LIN {X 0,Y 391.58,Z 838.555,A -85,B 0,C 180,E1 -11591.925,E2 -11591.925} C_VEL
LIN {X 0,Y 392.931,Z 851.436,A -85,B 0,C 180,E1 -11592.757,E2 -11592.757} C_VEL
LIN {X 0,Y 393.603,Z 859.87,A -85,B 0,C 180,E1 -11593.4,E2 -11593.4} C_VEL
LIN {X 0,Y 392.572,Z 872.076,A -85,B 0,C 180,E1 -11594.423,E2 -11594.423} C_VEL
LIN {X 0,Y 391.606,Z 884.787,A -85,B 0,C 180,E1 -11595.726,E2 -11595.726} C_VEL
LIN {X 0,Y 390.818,Z 894.925,A -85,B 0,C 180,E1 -11597.01,E2 -11597.01} C_VEL
LIN {X 0,Y 390.076,Z 904.821,A -85,B 0,C 180,E1 -11598.569,E2 -11598.569} C_VEL
LIN {X 0,Y 389.501,Z 912.81,A -85,B 0,C 180,E1 -11600.13,E2 -11600.13} C_VEL
LIN {X 0,Y 389.129,Z 919.186,A -85,B 0,C 180,E1 -11601.692,E2 -11601.692} C_VEL
LIN {X 0,Y 388.914,Z 924.388,A -85,B 0,C 180,E1 -11603.307,E2 -11603.307} C_VEL
LIN {X 0,Y 388.848,Z 928.132,A -85,B 0,C 180,E1 -11604.815,E2 -11604.815} C_VEL
LIN {X 0,Y 388.745,Z 930.111,A -85,B 0,C 180,E1 -11605.853,E2 -11605.853} C_VEL
LIN {X 0,Y 388.737,Z 931.665,A -85,B 0,C 180,E1 -11606.891,E2 -11606.891} C_VEL
LIN {X 0,Y 388.832,Z 932.76,A -85,B 0,C 180,E1 -11607.928,E2 -11607.928} C_VEL
LIN {X 0,Y 388.809,Z 933.409,A -85,B 0,C 180,E1 -11608.964,E2 -11608.964} C_VEL
LIN {X 0,Y 388.823,Z 933.651,A -85,B 0,C 180,E1 -11610,E2 -11610} C_VEL
LIN {X 0,Y 388.809,Z 933.483,A -85,B 0,C 180,E1 -11611.036,E2 -11611.036} C_VEL
LIN {X 0,Y 388.836,Z 932.855,A -85,B 0,C 180,E1 -11612.072,E2 -11612.072} C_VEL
LIN {X 0,Y 388.757,Z 930.333,A -85,B 0,C 180,E1 -11614.147,E2 -11614.147} C_VEL
LIN {X 0,Y 388.817,Z 926.891,A -85,B 0,C 180,E1 -11615.88,E2 -11615.88} C_VEL
LIN {X 0,Y 388.95,Z 923.164,A -85,B 0,C 180,E1 -11617.267,E2 -11617.267} C_VEL
LIN {X 0,Y 389.305,Z 916.887,A -85,B 0,C 180,E1 -11619.089,E2 -11619.089} C_VEL
LIN {X 0,Y 389.747,Z 910.033,A -85,B 0,C 180,E1 -11620.651,E2 -11620.651} C_VEL
LIN {X 0,Y 390.464,Z 901.593,A -85,B 0,C 180,E1 -11622.21,E2 -11622.21} C_VEL
LIN {X 0,Y 391.331,Z 891.841,A -85,B 0,C 180,E1 -11623.68,E2 -11623.68} C_VEL
LIN {X 0,Y 392.274,Z 880.534,A -85,B 0,C 180,E1 -11625.057,E2 -11625.057} C_VEL
LIN {X 0,Y 393.418,Z 868.68,A -85,B 0,C 180,E1 -11626.208,E2 -11626.208} C_VEL
LIN {X 0,Y 394.056,Z 859.025,A -85,B 0,C 180,E1 -11626.981,E2 -11626.981} C_VEL
LIN {X 0,Y 393.075,Z 845.103,A -85,B 0,C 180,E1 -11627.969,E2 -11627.969} C_VEL
LIN {X 0,Y 391.432,Z 832.806,A -85,B 0,C 180,E1 -11628.703,E2 -11628.703} C_VEL
LIN {X 0,Y 389.433,Z 823.338,A -85,B 0,C 180,E1 -11629.23,E2 -11629.23} C_VEL
LIN {X 0,Y 389.856,Z 815.289,A -85,B 0,C 180,E1 -11632.716,E2 -11632.716} C_VEL
LIN {X 0,Y 390.344,Z 808.49,A -85,B 0,C 180,E1 -11635.81,E2 -11635.81} C_VEL
LIN {X 0,Y 390.913,Z 801.858,A -85,B 0,C 180,E1 -11639.04,E2 -11639.04} C_VEL
LIN {X 0,Y 391.767,Z 795.266,A -85,B 0,C 180,E1 -11642.56,E2 -11642.56} C_VEL
LIN {X 0,Y 392.323,Z 791.243,A -85,B 0,C 180,E1 -11644.977,E2 -11644.977} C_VEL
LIN {X 0,Y 392.483,Z 787.628,A -85,B 0,C 180,E1 -11647.505,E2 -11647.505} C_VEL
LIN {X 0,Y 392.083,Z 784.529,A -85,B 0,C 180,E1 -11650.188,E2 -11650.188} C_VEL
LIN {X 0,Y 391.699,Z 782.043,A -85,B 0,C 180,E1 -11652.985,E2 -11652.985} C_VEL
LIN {X 0,Y 391.348,Z 780.234,A -85,B 0,C 180,E1 -11655.918,E2 -11655.918} C_VEL
LIN {X 0,Y 391.117,Z 779.149,A -85,B 0,C 180,E1 -11658.999,E2 -11658.999} C_VEL
LIN {X 0,Y 391.069,Z 778.836,A -85,B 0,C 180,E1 -11661.023,E2 -11661.023} C_VEL
LIN {X 0,Y 390.893,Z 778.937,A -85,B 0,C 180,E1 -11664.006,E2 -11664.006} C_VEL
LIN {X 0,Y 390.778,Z 779.326,A -85,B 0,C 180,E1 -11666.114,E2 -11666.114} C_VEL
LIN {X 0,Y 390.508,Z 780.09,A -85,B 0,C 180,E1 -11668.538,E2 -11668.538} C_VEL
LIN {X 0,Y 390.157,Z 781.62,A -85,B 0,C 180,E1 -11672.072,E2 -11672.072} C_VEL
LIN {X 0,Y 389.86,Z 783.496,A -85,B 0,C 180,E1 -11675.504,E2 -11675.504} C_VEL
LIN {X 0,Y 389.639,Z 785.619,A -85,B 0,C 180,E1 -11678.853,E2 -11678.853} C_VEL
LIN {X 0,Y 389.514,Z 787.117,A -85,B 0,C 180,E1 -11680.962,E2 -11680.962} C_VEL
LIN {X 0,Y 393.71,Z 799.562,A -85,B 0,C 180,E1 -11681.858,E2 -11681.858} C_VEL
LIN {X 0,Y 395.904,Z 808.974,A -85,B 0,C 180,E1 -11682.582,E2 -11682.582} C_VEL
LIN {X 0,Y 394.972,Z 821.103,A -85,B 0,C 180,E1 -11683.458,E2 -11683.458} C_VEL
LIN {X 0,Y 394.076,Z 832.258,A -85,B 0,C 180,E1 -11684.483,E2 -11684.483} C_VEL
LIN {X 0,Y 393.023,Z 843.465,A -85,B 0,C 180,E1 -11685.765,E2 -11685.765} C_VEL
LIN {X 0,Y 392.055,Z 852.61,A -85,B 0,C 180,E1 -11687.05,E2 -11687.05} C_VEL
LIN {X 0,Y 391.22,Z 861.469,A -85,B 0,C 180,E1 -11688.602,E2 -11688.602} C_VEL
LIN {X 0,Y 390.495,Z 868.618,A -85,B 0,C 180,E1 -11690.154,E2 -11690.154} C_VEL
LIN {X 0,Y 389.9,Z 874.374,A -85,B 0,C 180,E1 -11691.708,E2 -11691.708} C_VEL
LIN {X 0,Y 389.555,Z 878.773,A -85,B 0,C 180,E1 -11693.215,E2 -11693.215} C_VEL
LIN {X 0,Y 389.112,Z 882.348,A -85,B 0,C 180,E1 -11694.818,E2 -11694.818} C_VEL
LIN {X 0,Y 389.158,Z 884.056,A -85,B 0,C 180,E1 -11695.856,E2 -11695.856} C_VEL
LIN {X 0,Y 389.016,Z 885.331,A -85,B 0,C 180,E1 -11696.892,E2 -11696.892} C_VEL
LIN {X 0,Y 388.923,Z 886.208,A -85,B 0,C 180,E1 -11697.928,E2 -11697.928} C_VEL
LIN {X 0,Y 388.862,Z 886.689,A -85,B 0,C 180,E1 -11698.963,E2 -11698.963} C_VEL
LIN {X 0,Y 388.823,Z 886.73,A -85,B 0,C 180,E1 -11699.999,E2 -11699.999} C_VEL
LIN {X 0,Y 388.837,Z 886.362,A -85,B 0,C 180,E1 -11701.035,E2 -11701.035} C_VEL
LIN {X 0,Y 388.898,Z 885.6,A -85,B 0,C 180,E1 -11702.07,E2 -11702.07} C_VEL
LIN {X 0,Y 388.96,Z 884.434,A -85,B 0,C 180,E1 -11703.106,E2 -11703.106} C_VEL
LIN {X 0,Y 388.965,Z 881.862,A -85,B 0,C 180,E1 -11704.663,E2 -11704.663} C_VEL
LIN {X 0,Y 389.259,Z 878.257,A -85,B 0,C 180,E1 -11706.218,E2 -11706.218} C_VEL
LIN {X 0,Y 389.458,Z 873.538,A -85,B 0,C 180,E1 -11707.777,E2 -11707.777} C_VEL
LIN {X 0,Y 389.915,Z 867.546,A -85,B 0,C 180,E1 -11709.335,E2 -11709.335} C_VEL
LIN {X 0,Y 390.483,Z 860.089,A -85,B 0,C 180,E1 -11710.892,E2 -11710.892} C_VEL
LIN {X 0,Y 391.195,Z 850.868,A -85,B 0,C 180,E1 -11712.449,E2 -11712.449} C_VEL
LIN {X 0,Y 392.147,Z 840.272,A -85,B 0,C 180,E1 -11713.868,E2 -11713.868} C_VEL
LIN {X 0,Y 392.862,Z 828.851,A -85,B 0,C 180,E1 -11715.105,E2 -11715.105} C_VEL
LIN {X 0,Y 393.588,Z 817.632,A -85,B 0,C 180,E1 -11716.066,E2 -11716.066} C_VEL
LIN {X 0,Y 394.225,Z 807.061,A -85,B 0,C 180,E1 -11716.789,E2 -11716.789} C_VEL
LIN {X 0,Y 391.983,Z 795.795,A -85,B 0,C 180,E1 -11717.5,E2 -11717.5} C_VEL
LIN {X 0,Y 388.944,Z 782.751,A -85,B 0,C 180,E1 -11718.16,E2 -11718.16} C_VEL
LIN {X 0,Y 388.983,Z 779.744,A -85,B 0,C 180,E1 -11721.182,E2 -11721.182} C_VEL
LIN {X 0,Y 389.066,Z 776.45,A -85,B 0,C 180,E1 -11724.547,E2 -11724.547} C_VEL
LIN {X 0,Y 389.164,Z 773.381,A -85,B 0,C 180,E1 -11727.76,E2 -11727.76} C_VEL
LIN {X 0,Y 389.428,Z 772.979,A -85,B 0,C 180,E1 -11730.351,E2 -11730.351} C_VEL
LIN {X 0,Y 389.737,Z 772.939,A -85,B 0,C 180,E1 -11732.749,E2 -11732.749} C_VEL
LIN {X 0,Y 389.97,Z 772.907,A -85,B 0,C 180,E1 -11735.807,E2 -11735.807} C_VEL
LIN {X 0,Y 390.064,Z 772.896,A -85,B 0,C 180,E1 -11739.217,E2 -11739.217} C_VEL
LIN {X 0,Y 390.038,Z 772.9,A -85,B 0,C 180,E1 -11742.373,E2 -11742.373} C_VEL
LIN {X 0,Y 390.039,Z 772.899,A -85,B 0,C 180,E1 -11745.353,E2 -11745.353} C_VEL
LIN {X 0,Y 390.025,Z 772.901,A -85,B 0,C 180,E1 -11748.186,E2 -11748.186} C_VEL
LIN {X 0,Y 390.082,Z 772.896,A -85,B 0,C 180,E1 -11750.906,E2 -11750.906} C_VEL
LIN {X 0,Y 390.077,Z 772.895,A -85,B 0,C 180,E1 -11754.792,E2 -11754.792} C_VEL
LIN {X 0,Y 390.015,Z 772.901,A -85,B 0,C 180,E1 -11758.495,E2 -11758.495} C_VEL
LIN {X 0,Y 390.031,Z 772.898,A -85,B 0,C 180,E1 -11762.063,E2 -11762.063} C_VEL
LIN {X 0,Y 390.052,Z 772.901,A -85,B 0,C 180,E1 -11765.517,E2 -11765.517} C_VEL
LIN {X 0,Y 390.047,Z 772.897,A -85,B 0,C 180,E1 -11768.877,E2 -11768.877} C_VEL
LIN {X 0,Y 390.102,Z 772.89,A -85,B 0,C 180,E1 -11772.165,E2 -11772.165} C_VEL
LIN {X 0,Y 390.134,Z 772.888,A -85,B 0,C 180,E1 -11775.392,E2 -11775.392} C_VEL
LIN {X 0,Y 390.135,Z 772.885,A -85,B 0,C 180,E1 -11778.571,E2 -11778.571} C_VEL
LIN {X 0,Y 390.246,Z 772.874,A -85,B 0,C 180,E1 -11782.086,E2 -11782.086} C_VEL
LIN {X 0,Y 390.188,Z 772.878,A -85,B 0,C 180,E1 -11784.833,E2 -11784.833} C_VEL
LIN {X 0,Y 390.396,Z 772.858,A -85,B 0,C 180,E1 -11787.937,E2 -11787.937} C_VEL
LIN {X 0,Y 390.392,Z 772.859,A -85,B 0,C 180,E1 -11792.063,E2 -11792.063} C_VEL
LIN {X 0,Y 390.264,Z 772.875,A -85,B 0,C 180,E1 -11796.203,E2 -11796.203} C_VEL
LIN {X 0,Y 390.174,Z 772.879,A -85,B 0,C 180,E1 -11799.33,E2 -11799.33} C_VEL
LIN {X 0,Y 390.185,Z 772.878,A -85,B 0,C 180,E1 -11803.439,E2 -11803.439} C_VEL
LIN {X 0,Y 390.12,Z 772.887,A -85,B 0,C 180,E1 -11807.299,E2 -11807.299} C_VEL
LIN {X 0,Y 390.079,Z 772.898,A -85,B 0,C 180,E1 -11810.471,E2 -11810.471} C_VEL
LIN {X 0,Y 390.056,Z 772.895,A -85,B 0,C 180,E1 -11813.353,E2 -11813.353} C_VEL
LIN {X 0,Y 390.04,Z 772.901,A -85,B 0,C 180,E1 -11816.807,E2 -11816.807} C_VEL
LIN {X 0,Y 389.332,Z 772.985,A -85,B 0,C 180,E1 -11817.669,E2 -11817.669} C_VEL
LIN {X 0,Y 386.463,Z 773.345,A -85,B 0,C 180,E1 -11819.07,E2 -11819.07} C_VEL
LIN {X 0,Y 384.063,Z 773.645,A -85,B 0,C 180,E1 -11820.203,E2 -11820.203} C_VEL
LIN {X 0,Y 383.043,Z 773.772,A -85,B 0,C 180,E1 -11821.079,E2 -11821.079} C_VEL
LIN {X 0,Y 382.963,Z 773.779,A -85,B 0,C 180,E1 -11821.375,E2 -11821.375} C_VEL
LIN {X 0,Y 383.011,Z 773.776,A -85,B 0,C 180,E1 -11824.669,E2 -11824.669} C_VEL
LIN {X 0,Y 382.992,Z 773.775,A -85,B 0,C 180,E1 -11827.905,E2 -11827.905} C_VEL
LIN {X 0,Y 382.978,Z 773.78,A -85,B 0,C 180,E1 -11831.348,E2 -11831.348} C_VEL
LIN {X 0,Y 382.99,Z 773.776,A -85,B 0,C 180,E1 -11834.304,E2 -11834.304} C_VEL
LIN {X 0,Y 383.005,Z 773.778,A -85,B 0,C 180,E1 -11837.241,E2 -11837.241} C_VEL
LIN {X 0,Y 383.01,Z 773.773,A -85,B 0,C 180,E1 -11840.415,E2 -11840.415} C_VEL
LIN {X 0,Y 382.955,Z 773.782,A -85,B 0,C 180,E1 -11844.039,E2 -11844.039} C_VEL
LIN {X 0,Y 382.762,Z 773.805,A -85,B 0,C 180,E1 -11846.577,E2 -11846.577} C_VEL
LIN {X 0,Y 382.408,Z 773.854,A -85,B 0,C 180,E1 -11849.744,E2 -11849.744} C_VEL
LIN {X 0,Y 382.057,Z 773.896,A -85,B 0,C 180,E1 -11852.622,E2 -11852.622} C_VEL
LIN {X 0,Y 381.957,Z 774.358,A -85,B 0,C 180,E1 -11853.795,E2 -11853.795} C_VEL
LIN {X 0,Y 381.905,Z 778.018,A -85,B 0,C 180,E1 -11857.267,E2 -11857.267} C_VEL
LIN {X 0,Y 381.859,Z 781.611,A -85,B 0,C 180,E1 -11860.655,E2 -11860.655} C_VEL
LIN {X 0,Y 381.864,Z 782.834,A -85,B 0,C 180,E1 -11861.717,E2 -11861.717} C_VEL
LIN {X 0,Y 384.853,Z 796.061,A -85,B 0,C 180,E1 -11862.369,E2 -11862.369} C_VEL
LIN {X 0,Y 387.203,Z 807.715,A -85,B 0,C 180,E1 -11863.119,E2 -11863.119} C_VEL
LIN {X 0,Y 386.421,Z 820.405,A -85,B 0,C 180,E1 -11864.034,E2 -11864.034} C_VEL
LIN {X 0,Y 385.715,Z 831.457,A -85,B 0,C 180,E1 -11865.051,E2 -11865.051} C_VEL
LIN {X 0,Y 384.861,Z 843.14,A -85,B 0,C 180,E1 -11866.403,E2 -11866.403} C_VEL
LIN {X 0,Y 384.098,Z 851.523,A -85,B 0,C 180,E1 -11867.586,E2 -11867.586} C_VEL
LIN {X 0,Y 383.392,Z 860.682,A -85,B 0,C 180,E1 -11869.171,E2 -11869.171} C_VEL
LIN {X 0,Y 382.773,Z 868.063,A -85,B 0,C 180,E1 -11870.756,E2 -11870.756} C_VEL
LIN {X 0,Y 382.407,Z 873.084,A -85,B 0,C 180,E1 -11872.078,E2 -11872.078} C_VEL
LIN {X 0,Y 382.187,Z 877.955,A -85,B 0,C 180,E1 -11873.667,E2 -11873.667} C_VEL
LIN {X 0,Y 381.884,Z 881.694,A -85,B 0,C 180,E1 -11875.251,E2 -11875.251} C_VEL
LIN {X 0,Y 381.842,Z 884.389,A -85,B 0,C 180,E1 -11876.836,E2 -11876.836} C_VEL
LIN {X 0,Y 381.822,Z 885.667,A -85,B 0,C 180,E1 -11877.891,E2 -11877.891} C_VEL
LIN {X 0,Y 381.755,Z 886.486,A -85,B 0,C 180,E1 -11878.946,E2 -11878.946} C_VEL
LIN {X 0,Y 381.777,Z 886.936,A -85,B 0,C 180,E1 -11881.056,E2 -11881.056} C_VEL
LIN {X 0,Y 381.837,Z 886.529,A -85,B 0,C 180,E1 -11882.111,E2 -11882.111} C_VEL
LIN {X 0,Y 381.952,Z 885.696,A -85,B 0,C 180,E1 -11883.165,E2 -11883.165} C_VEL
LIN {X 0,Y 382.092,Z 884.467,A -85,B 0,C 180,E1 -11884.22,E2 -11884.22} C_VEL
LIN {X 0,Y 382.157,Z 881.821,A -85,B 0,C 180,E1 -11885.806,E2 -11885.806} C_VEL
LIN {X 0,Y 382.595,Z 878.139,A -85,B 0,C 180,E1 -11887.389,E2 -11887.389} C_VEL
LIN {X 0,Y 383.055,Z 873.344,A -85,B 0,C 180,E1 -11888.973,E2 -11888.973} C_VEL
LIN {X 0,Y 383.676,Z 867.268,A -85,B 0,C 180,E1 -11890.556,E2 -11890.556} C_VEL
LIN {X 0,Y 384.548,Z 859.668,A -85,B 0,C 180,E1 -11892.134,E2 -11892.134} C_VEL
LIN {X 0,Y 385.437,Z 850.314,A -85,B 0,C 180,E1 -11893.713,E2 -11893.713} C_VEL
LIN {X 0,Y 386.64,Z 840.208,A -85,B 0,C 180,E1 -11895.067,E2 -11895.067} C_VEL
LIN {X 0,Y 387.525,Z 830.053,A -85,B 0,C 180,E1 -11896.192,E2 -11896.192} C_VEL
LIN {X 0,Y 388.598,Z 818.241,A -85,B 0,C 180,E1 -11897.228,E2 -11897.228} C_VEL
LIN {X 0,Y 389.197,Z 811.105,A -85,B 0,C 180,E1 -11897.742,E2 -11897.742} C_VEL
LIN {X 0,Y 388.265,Z 805.179,A -85,B 0,C 180,E1 -11898.212,E2 -11898.212} C_VEL
LIN {X 0,Y 385.085,Z 794.046,A -85,B 0,C 180,E1 -11899.081,E2 -11899.081} C_VEL
LIN {X 0,Y 382.431,Z 786.484,A -85,B 0,C 180,E1 -11899.632,E2 -11899.632} C_VEL
LIN {X 0,Y 382.479,Z 782.25,A -85,B 0,C 180,E1 -11903.845,E2 -11903.845} C_VEL
LIN {X 0,Y 382.586,Z 778.671,A -85,B 0,C 180,E1 -11907.339,E2 -11907.339} C_VEL
LIN {X 0,Y 382.647,Z 775.618,A -85,B 0,C 180,E1 -11910.317,E2 -11910.317} C_VEL
LIN {X 0,Y 382.633,Z 773.826,A -85,B 0,C 180,E1 -11912.338,E2 -11912.338} C_VEL
LIN {X 0,Y 382.852,Z 773.798,A -85,B 0,C 180,E1 -11914.686,E2 -11914.686} C_VEL
LIN {X 0,Y 382.998,Z 773.778,A -85,B 0,C 180,E1 -11917.903,E2 -11917.903} C_VEL
LIN {X 0,Y 382.986,Z 773.781,A -85,B 0,C 180,E1 -11921.348,E2 -11921.348} C_VEL
LIN {X 0,Y 383,Z 773.778,A -85,B 0,C 180,E1 -11924.304,E2 -11924.304} C_VEL
LIN {X 0,Y 383.029,Z 773.922,A -85,B 0,C 180,E1 -11925.887,E2 -11925.887} C_VEL
LIN {X 0,Y 383.975,Z 779.024,A -85,B 0,C 180,E1 -11928.782,E2 -11928.782} C_VEL
LIN {X 0,Y 384.932,Z 784.447,A -85,B 0,C 180,E1 -11931.73,E2 -11931.73} C_VEL
LIN {X 0,Y 385.321,Z 787.597,A -85,B 0,C 180,E1 -11933.374,E2 -11933.374} C_VEL
LIN {X 0,Y 385.109,Z 791.985,A -85,B 0,C 180,E1 -11935.547,E2 -11935.547} C_VEL
LIN {X 0,Y 384.339,Z 799.635,A -85,B 0,C 180,E1 -11939.202,E2 -11939.202} C_VEL
LIN {X 0,Y 383.564,Z 808.537,A -85,B 0,C 180,E1 -11943.326,E2 -11943.326} C_VEL
LIN {X 0,Y 382.988,Z 815.713,A -85,B 0,C 180,E1 -11946.568,E2 -11946.568} C_VEL
LIN {X 0,Y 382.532,Z 823.743,A -85,B 0,C 180,E1 -11950.13,E2 -11950.13} C_VEL
LIN {X 0,Y 382.427,Z 825.082,A -85,B 0,C 180,E1 -11950.718,E2 -11950.718} C_VEL
LIN {X 0,Y 384.716,Z 837.37,A -85,B 0,C 180,E1 -11951.432,E2 -11951.432} C_VEL
LIN {X 0,Y 386.051,Z 850.482,A -85,B 0,C 180,E1 -11952.307,E2 -11952.307} C_VEL
LIN {X 0,Y 386.834,Z 860.536,A -85,B 0,C 180,E1 -11953.101,E2 -11953.101} C_VEL
LIN {X 0,Y 385.747,Z 872.461,A -85,B 0,C 180,E1 -11954.14,E2 -11954.14} C_VEL
LIN {X 0,Y 384.728,Z 883.774,A -85,B 0,C 180,E1 -11955.379,E2 -11955.379} C_VEL
LIN {X 0,Y 383.865,Z 894.061,A -85,B 0,C 180,E1 -11956.77,E2 -11956.77} C_VEL
LIN {X 0,Y 383.084,Z 904.033,A -85,B 0,C 180,E1 -11958.357,E2 -11958.357} C_VEL
LIN {X 0,Y 382.468,Z 912.088,A -85,B 0,C 180,E1 -11959.947,E2 -11959.947} C_VEL
LIN {X 0,Y 382.06,Z 918.54,A -85,B 0,C 180,E1 -11961.538,E2 -11961.538} C_VEL
LIN {X 0,Y 381.844,Z 923.648,A -85,B 0,C 180,E1 -11963.129,E2 -11963.129} C_VEL
LIN {X 0,Y 381.763,Z 927.58,A -85,B 0,C 180,E1 -11964.719,E2 -11964.719} C_VEL
LIN {X 0,Y 381.673,Z 929.58,A -85,B 0,C 180,E1 -11965.776,E2 -11965.776} C_VEL
LIN {X 0,Y 381.647,Z 931.148,A -85,B 0,C 180,E1 -11966.833,E2 -11966.833} C_VEL
LIN {X 0,Y 381.763,Z 932.279,A -85,B 0,C 180,E1 -11967.89,E2 -11967.89} C_VEL
LIN {X 0,Y 381.738,Z 932.941,A -85,B 0,C 180,E1 -11968.945,E2 -11968.945} C_VEL
LIN {X 0,Y 381.748,Z 933.199,A -85,B 0,C 180,E1 -11970,E2 -11970} C_VEL
LIN {X 0,Y 381.739,Z 933.044,A -85,B 0,C 180,E1 -11971.055,E2 -11971.055} C_VEL
LIN {X 0,Y 381.749,Z 932.448,A -85,B 0,C 180,E1 -11972.11,E2 -11972.11} C_VEL
LIN {X 0,Y 381.651,Z 931.407,A -85,B 0,C 180,E1 -11973.167,E2 -11973.167} C_VEL
LIN {X 0,Y 381.682,Z 929.957,A -85,B 0,C 180,E1 -11974.224,E2 -11974.224} C_VEL
LIN {X 0,Y 381.719,Z 926.892,A -85,B 0,C 180,E1 -11975.83,E2 -11975.83} C_VEL
LIN {X 0,Y 381.876,Z 922.84,A -85,B 0,C 180,E1 -11977.402,E2 -11977.402} C_VEL
LIN {X 0,Y 382.244,Z 916.613,A -85,B 0,C 180,E1 -11979.258,E2 -11979.258} C_VEL
LIN {X 0,Y 382.716,Z 909.836,A -85,B 0,C 180,E1 -11980.849,E2 -11980.849} C_VEL
LIN {X 0,Y 383.501,Z 901.502,A -85,B 0,C 180,E1 -11982.435,E2 -11982.435} C_VEL
LIN {X 0,Y 384.281,Z 893.091,A -85,B 0,C 180,E1 -11983.754,E2 -11983.754} C_VEL
LIN {X 0,Y 385.22,Z 882.965,A -85,B 0,C 180,E1 -11985.069,E2 -11985.069} C_VEL
LIN {X 0,Y 386.482,Z 870.482,A -85,B 0,C 180,E1 -11986.371,E2 -11986.371} C_VEL
LIN {X 0,Y 387.322,Z 861.364,A -85,B 0,C 180,E1 -11987.149,E2 -11987.149} C_VEL
LIN {X 0,Y 386.586,Z 848.495,A -85,B 0,C 180,E1 -11988.146,E2 -11988.146} C_VEL
LIN {X 0,Y 385.21,Z 835.852,A -85,B 0,C 180,E1 -11988.957,E2 -11988.957} C_VEL
LIN {X 0,Y 382.407,Z 822.757,A -85,B 0,C 180,E1 -11989.737,E2 -11989.737} C_VEL
LIN {X 0,Y 382.899,Z 814.56,A -85,B 0,C 180,E1 -11993.401,E2 -11993.401} C_VEL
LIN {X 0,Y 383.436,Z 807.64,A -85,B 0,C 180,E1 -11996.684,E2 -11996.684} C_VEL
LIN {X 0,Y 384.122,Z 800.834,A -85,B 0,C 180,E1 -12000.171,E2 -12000.171} C_VEL
LIN {X 0,Y 384.955,Z 795.443,A -85,B 0,C 180,E1 -12003.21,E2 -12003.21} C_VEL
LIN {X 0,Y 385.419,Z 791.549,A -85,B 0,C 180,E1 -12005.698,E2 -12005.698} C_VEL
LIN {X 0,Y 385.522,Z 789.755,A -85,B 0,C 180,E1 -12006.984,E2 -12006.984} C_VEL
LIN {X 0,Y 385.454,Z 788.025,A -85,B 0,C 180,E1 -12008.369,E2 -12008.369} C_VEL
LIN {X 0,Y 384.961,Z 784.778,A -85,B 0,C 180,E1 -12011.537,E2 -12011.537} C_VEL
LIN {X 0,Y 384.578,Z 782.538,A -85,B 0,C 180,E1 -12014.543,E2 -12014.543} C_VEL
LIN {X 0,Y 384.287,Z 781.151,A -85,B 0,C 180,E1 -12017.415,E2 -12017.415} C_VEL
LIN {X 0,Y 384.142,Z 780.429,A -85,B 0,C 180,E1 -12020.211,E2 -12020.211} C_VEL
LIN {X 0,Y 384.009,Z 780.281,A -85,B 0,C 180,E1 -12022.845,E2 -12022.845} C_VEL
LIN {X 0,Y 383.853,Z 780.572,A -85,B 0,C 180,E1 -12025.478,E2 -12025.478} C_VEL
LIN {X 0,Y 383.616,Z 781.199,A -85,B 0,C 180,E1 -12027.906,E2 -12027.906} C_VEL
LIN {X 0,Y 383.165,Z 782.684,A -85,B 0,C 180,E1 -12031.693,E2 -12031.693} C_VEL
LIN {X 0,Y 382.899,Z 784.386,A -85,B 0,C 180,E1 -12035.028,E2 -12035.028} C_VEL
LIN {X 0,Y 382.657,Z 786.445,A -85,B 0,C 180,E1 -12038.448,E2 -12038.448} C_VEL
LIN {X 0,Y 382.551,Z 787.774,A -85,B 0,C 180,E1 -12040.444,E2 -12040.444} C_VEL
LIN {X 0,Y 386.649,Z 799.572,A -85,B 0,C 180,E1 -12041.346,E2 -12041.346} C_VEL
LIN {X 0,Y 389.098,Z 808.956,A -85,B 0,C 180,E1 -12042.117,E2 -12042.117} C_VEL
LIN {X 0,Y 389.2,Z 812.717,A -85,B 0,C 180,E1 -12042.393,E2 -12042.393} C_VEL
LIN {X 0,Y 388.226,Z 824.283,A -85,B 0,C 180,E1 -12043.298,E2 -12043.298} C_VEL
LIN {X 0,Y 387.167,Z 835.554,A -85,B 0,C 180,E1 -12044.412,E2 -12044.412} C_VEL
LIN {X 0,Y 386.234,Z 844.631,A -85,B 0,C 180,E1 -12045.51,E2 -12045.51} C_VEL
LIN {X 0,Y 385.225,Z 853.592,A -85,B 0,C 180,E1 -12046.817,E2 -12046.817} C_VEL
LIN {X 0,Y 384.324,Z 862.352,A -85,B 0,C 180,E1 -12048.395,E2 -12048.395} C_VEL
LIN {X 0,Y 383.553,Z 869.439,A -85,B 0,C 180,E1 -12049.974,E2 -12049.974} C_VEL
LIN {X 0,Y 382.931,Z 875.12,A -85,B 0,C 180,E1 -12051.556,E2 -12051.556} C_VEL
LIN {X 0,Y 382.522,Z 879.62,A -85,B 0,C 180,E1 -12053.159,E2 -12053.159} C_VEL
LIN {X 0,Y 382.062,Z 882.95,A -85,B 0,C 180,E1 -12054.722,E2 -12054.722} C_VEL
LIN {X 0,Y 382.11,Z 884.615,A -85,B 0,C 180,E1 -12055.78,E2 -12055.78} C_VEL
LIN {X 0,Y 381.965,Z 885.867,A -85,B 0,C 180,E1 -12056.835,E2 -12056.835} C_VEL
LIN {X 0,Y 381.858,Z 886.72,A -85,B 0,C 180,E1 -12057.889,E2 -12057.889} C_VEL
LIN {X 0,Y 381.79,Z 887.169,A -85,B 0,C 180,E1 -12058.944,E2 -12058.944} C_VEL
LIN {X 0,Y 381.749,Z 887.172,A -85,B 0,C 180,E1 -12059.999,E2 -12059.999} C_VEL
LIN {X 0,Y 381.766,Z 886.776,A -85,B 0,C 180,E1 -12061.054,E2 -12061.054} C_VEL
LIN {X 0,Y 381.833,Z 885.982,A -85,B 0,C 180,E1 -12062.109,E2 -12062.109} C_VEL
LIN {X 0,Y 381.869,Z 884.767,A -85,B 0,C 180,E1 -12063.164,E2 -12063.164} C_VEL
LIN {X 0,Y 381.899,Z 882.139,A -85,B 0,C 180,E1 -12064.749,E2 -12064.749} C_VEL
LIN {X 0,Y 382.199,Z 878.474,A -85,B 0,C 180,E1 -12066.333,E2 -12066.333} C_VEL
LIN {X 0,Y 382.408,Z 873.682,A -85,B 0,C 180,E1 -12067.922,E2 -12067.922} C_VEL
LIN {X 0,Y 382.989,Z 866.476,A -85,B 0,C 180,E1 -12069.772,E2 -12069.772} C_VEL
LIN {X 0,Y 383.635,Z 858.694,A -85,B 0,C 180,E1 -12071.357,E2 -12071.357} C_VEL
LIN {X 0,Y 384.421,Z 848.957,A -85,B 0,C 180,E1 -12072.94,E2 -12072.94} C_VEL
LIN {X 0,Y 385.315,Z 838.988,A -85,B 0,C 180,E1 -12074.254,E2 -12074.254} C_VEL
LIN {X 0,Y 386.032,Z 827.649,A -85,B 0,C 180,E1 -12075.458,E2 -12075.458} C_VEL
LIN {X 0,Y 386.831,Z 815.415,A -85,B 0,C 180,E1 -12076.491,E2 -12076.491} C_VEL
LIN {X 0,Y 387.327,Z 807.893,A -85,B 0,C 180,E1 -12076.999,E2 -12076.999} C_VEL
LIN {X 0,Y 384.733,Z 795.59,A -85,B 0,C 180,E1 -12077.79,E2 -12077.79} C_VEL
LIN {X 0,Y 381.881,Z 783.107,A -85,B 0,C 180,E1 -12078.439,E2 -12078.439} C_VEL
LIN {X 0,Y 381.933,Z 779.984,A -85,B 0,C 180,E1 -12081.592,E2 -12081.592} C_VEL
LIN {X 0,Y 382.054,Z 776.669,A -85,B 0,C 180,E1 -12085.029,E2 -12085.029} C_VEL
LIN {X 0,Y 382.132,Z 773.888,A -85,B 0,C 180,E1 -12088.018,E2 -12088.018} C_VEL
LIN {X 0,Y 382.46,Z 773.844,A -85,B 0,C 180,E1 -12090.964,E2 -12090.964} C_VEL
LIN {X 0,Y 382.829,Z 773.801,A -85,B 0,C 180,E1 -12094.298,E2 -12094.298} C_VEL
LIN {X 0,Y 382.975,Z 773.778,A -85,B 0,C 180,E1 -12097.269,E2 -12097.269} C_VEL
LIN {X 0,Y 383.004,Z 773.775,A -85,B 0,C 180,E1 -12099.957,E2 -12099.957} C_VEL
LIN {X 0,Y 383,Z 773.778,A -85,B 0,C 180,E1 -12102.777,E2 -12102.777} C_VEL
LIN {X 0,Y 382.992,Z 773.776,A -85,B 0,C 180,E1 -12105.788,E2 -12105.788} C_VEL
LIN {X 0,Y 382.982,Z 773.78,A -85,B 0,C 180,E1 -12108.795,E2 -12108.795} C_VEL
LIN {X 0,Y 382.992,Z 773.776,A -85,B 0,C 180,E1 -12112.095,E2 -12112.095} C_VEL
LIN {X 0,Y 383.011,Z 773.777,A -85,B 0,C 180,E1 -12115.331,E2 -12115.331} C_VEL
LIN {X 0,Y 382.974,Z 773.781,A -85,B 0,C 180,E1 -12119.08,E2 -12119.08} C_VEL
LIN {X 0,Y 382.985,Z 773.777,A -85,B 0,C 180,E1 -12122.692,E2 -12122.692} C_VEL
LIN {X 0,Y 383.008,Z 773.773,A -85,B 0,C 180,E1 -12126.191,E2 -12126.191} C_VEL
LIN {X 0,Y 383.047,Z 773.773,A -85,B 0,C 180,E1 -12129.598,E2 -12129.598} C_VEL
LIN {X 0,Y 383.085,Z 773.764,A -85,B 0,C 180,E1 -12132.93,E2 -12132.93} C_VEL
LIN {X 0,Y 383.116,Z 773.759,A -85,B 0,C 180,E1 -12136.464,E2 -12136.464} C_VEL
LIN {X 0,Y 383.132,Z 773.757,A -85,B 0,C 180,E1 -12140.497,E2 -12140.497} C_VEL
LIN {X 0,Y 383.223,Z 773.75,A -85,B 0,C 180,E1 -12143.683,E2 -12143.683} C_VEL
LIN {X 0,Y 383.362,Z 773.734,A -85,B 0,C 180,E1 -12147.899,E2 -12147.899} C_VEL
LIN {X 0,Y 383.357,Z 773.735,A -85,B 0,C 180,E1 -12152.101,E2 -12152.101} C_VEL
LIN {X 0,Y 383.222,Z 773.75,A -85,B 0,C 180,E1 -12156.317,E2 -12156.317} C_VEL
LIN {X 0,Y 383.125,Z 773.758,A -85,B 0,C 180,E1 -12159.503,E2 -12159.503} C_VEL
LIN {X 0,Y 383.116,Z 773.759,A -85,B 0,C 180,E1 -12163.536,E2 -12163.536} C_VEL
LIN {X 0,Y 383.085,Z 773.764,A -85,B 0,C 180,E1 -12167.07,E2 -12167.07} C_VEL
LIN {X 0,Y 383.02,Z 773.776,A -85,B 0,C 180,E1 -12170.647,E2 -12170.647} C_VEL
LIN {X 0,Y 383.004,Z 773.773,A -85,B 0,C 180,E1 -12173.809,E2 -12173.809} C_VEL
LIN {X 0,Y 382.983,Z 773.777,A -85,B 0,C 180,E1 -12177.308,E2 -12177.308} C_VEL
LIN {X 0,Y 382.974,Z 773.781,A -85,B 0,C 180,E1 -12180.92,E2 -12180.92} C_VEL
LIN {X 0,Y 382.963,Z 773.779,A -85,B 0,C 180,E1 -12181.375,E2 -12181.375} C_VEL
LIN {X 0,Y 382.304,Z 773.863,A -85,B 0,C 180,E1 -12182.254,E2 -12182.254} C_VEL
LIN {X 0,Y 379.452,Z 774.216,A -85,B 0,C 180,E1 -12183.682,E2 -12183.682} C_VEL
LIN {X 0,Y 377.039,Z 774.522,A -85,B 0,C 180,E1 -12184.837,E2 -12184.837} C_VEL
LIN {X 0,Y 376.014,Z 774.645,A -85,B 0,C 180,E1 -12185.73,E2 -12185.73} C_VEL
LIN {X 0,Y 375.937,Z 774.654,A -85,B 0,C 180,E1 -12186.032,E2 -12186.032} C_VEL
LIN {X 0,Y 375.955,Z 774.654,A -85,B 0,C 180,E1 -12189.464,E2 -12189.464} C_VEL
LIN {X 0,Y 375.929,Z 774.659,A -85,B 0,C 180,E1 -12193.191,E2 -12193.191} C_VEL
LIN {X 0,Y 375.929,Z 774.657,A -85,B 0,C 180,E1 -12196.812,E2 -12196.812} C_VEL
LIN {X 0,Y 375.957,Z 774.652,A -85,B 0,C 180,E1 -12200.539,E2 -12200.539} C_VEL
LIN {X 0,Y 375.911,Z 774.661,A -85,B 0,C 180,E1 -12203.507,E2 -12203.507} C_VEL
LIN {X 0,Y 375.778,Z 774.678,A -85,B 0,C 180,E1 -12205.871,E2 -12205.871} C_VEL
LIN {X 0,Y 375.518,Z 774.707,A -85,B 0,C 180,E1 -12208.398,E2 -12208.398} C_VEL
LIN {X 0,Y 375.092,Z 774.764,A -85,B 0,C 180,E1 -12212.07,E2 -12212.07} C_VEL
LIN {X 0,Y 374.931,Z 774.785,A -85,B 0,C 180,E1 -12213.266,E2 -12213.266} C_VEL
LIN {X 0,Y 374.889,Z 775.704,A -85,B 0,C 180,E1 -12214.459,E2 -12214.459} C_VEL
LIN {X 0,Y 374.813,Z 779.418,A -85,B 0,C 180,E1 -12217.976,E2 -12217.976} C_VEL
LIN {X 0,Y 374.807,Z 783.107,A -85,B 0,C 180,E1 -12221.443,E2 -12221.443} C_VEL
LIN {X 0,Y 377.658,Z 795.915,A -85,B 0,C 180,E1 -12222.088,E2 -12222.088} C_VEL
LIN {X 0,Y 380.231,Z 808.802,A -85,B 0,C 180,E1 -12222.938,E2 -12222.938} C_VEL
LIN {X 0,Y 379.446,Z 821.333,A -85,B 0,C 180,E1 -12223.871,E2 -12223.871} C_VEL
LIN {X 0,Y 378.717,Z 832.579,A -85,B 0,C 180,E1 -12224.943,E2 -12224.943} C_VEL
LIN {X 0,Y 377.849,Z 843.865,A -85,B 0,C 180,E1 -12226.283,E2 -12226.283} C_VEL
LIN {X 0,Y 377.02,Z 853.036,A -85,B 0,C 180,E1 -12227.623,E2 -12227.623} C_VEL
LIN {X 0,Y 376.28,Z 861.981,A -85,B 0,C 180,E1 -12229.237,E2 -12229.237} C_VEL
LIN {X 0,Y 375.671,Z 869.223,A -85,B 0,C 180,E1 -12230.851,E2 -12230.851} C_VEL
LIN {X 0,Y 375.237,Z 874.998,A -85,B 0,C 180,E1 -12232.468,E2 -12232.468} C_VEL
LIN {X 0,Y 375.037,Z 879.538,A -85,B 0,C 180,E1 -12234.085,E2 -12234.085} C_VEL
LIN {X 0,Y 374.769,Z 882.984,A -85,B 0,C 180,E1 -12235.699,E2 -12235.699} C_VEL
LIN {X 0,Y 374.752,Z 884.706,A -85,B 0,C 180,E1 -12236.776,E2 -12236.776} C_VEL
LIN {X 0,Y 374.758,Z 886.02,A -85,B 0,C 180,E1 -12237.852,E2 -12237.852} C_VEL
LIN {X 0,Y 374.686,Z 886.884,A -85,B 0,C 180,E1 -12238.926,E2 -12238.926} C_VEL
LIN {X 0,Y 374.656,Z 887.335,A -85,B 0,C 180,E1 -12240.001,E2 -12240.001} C_VEL
LIN {X 0,Y 374.707,Z 887.388,A -85,B 0,C 180,E1 -12241.076,E2 -12241.076} C_VEL
LIN {X 0,Y 374.776,Z 887.031,A -85,B 0,C 180,E1 -12242.15,E2 -12242.15} C_VEL
LIN {X 0,Y 374.903,Z 886.229,A -85,B 0,C 180,E1 -12243.225,E2 -12243.225} C_VEL
LIN {X 0,Y 375.044,Z 885.034,A -85,B 0,C 180,E1 -12244.3,E2 -12244.3} C_VEL
LIN {X 0,Y 375.127,Z 882.452,A -85,B 0,C 180,E1 -12245.915,E2 -12245.915} C_VEL
LIN {X 0,Y 375.583,Z 878.823,A -85,B 0,C 180,E1 -12247.528,E2 -12247.528} C_VEL
LIN {X 0,Y 376.101,Z 874.078,A -85,B 0,C 180,E1 -12249.14,E2 -12249.14} C_VEL
LIN {X 0,Y 376.859,Z 866.938,A -85,B 0,C 180,E1 -12251.021,E2 -12251.021} C_VEL
LIN {X 0,Y 377.839,Z 859.234,A -85,B 0,C 180,E1 -12252.625,E2 -12252.625} C_VEL
LIN {X 0,Y 378.631,Z 851.438,A -85,B 0,C 180,E1 -12253.964,E2 -12253.964} C_VEL
LIN {X 0,Y 379.912,Z 841.359,A -85,B 0,C 180,E1 -12255.355,E2 -12255.355} C_VEL
LIN {X 0,Y 380.81,Z 831.608,A -85,B 0,C 180,E1 -12256.471,E2 -12256.471} C_VEL
LIN {X 0,Y 381.987,Z 820.111,A -85,B 0,C 180,E1 -12257.535,E2 -12257.535} C_VEL
LIN {X 0,Y 382.654,Z 811.427,A -85,B 0,C 180,E1 -12258.195,E2 -12258.195} C_VEL
LIN {X 0,Y 380.775,Z 802.763,A -85,B 0,C 180,E1 -12258.927,E2 -12258.927} C_VEL
LIN {X 0,Y 376.631,Z 790.283,A -85,B 0,C 180,E1 -12259.947,E2 -12259.947} C_VEL
LIN {X 0,Y 375.423,Z 787.095,A -85,B 0,C 180,E1 -12260.204,E2 -12260.204} C_VEL
LIN {X 0,Y 375.506,Z 783.831,A -85,B 0,C 180,E1 -12263.495,E2 -12263.495} C_VEL
LIN {X 0,Y 375.572,Z 780.648,A -85,B 0,C 180,E1 -12266.687,E2 -12266.687} C_VEL
LIN {X 0,Y 375.644,Z 778.246,A -85,B 0,C 180,E1 -12269.108,E2 -12269.108} C_VEL
LIN {X 0,Y 375.65,Z 775.8,A -85,B 0,C 180,E1 -12271.592,E2 -12271.592} C_VEL
LIN {X 0,Y 375.65,Z 774.696,A -85,B 0,C 180,E1 -12272.859,E2 -12272.859} C_VEL
LIN {X 0,Y 375.864,Z 774.669,A -85,B 0,C 180,E1 -12275.427,E2 -12275.427} C_VEL
LIN {X 0,Y 375.972,Z 774.652,A -85,B 0,C 180,E1 -12278.27,E2 -12278.27} C_VEL
LIN {X 0,Y 375.937,Z 774.658,A -85,B 0,C 180,E1 -12281.601,E2 -12281.601} C_VEL
LIN {X 0,Y 375.942,Z 774.658,A -85,B 0,C 180,E1 -12285.394,E2 -12285.394} C_VEL
LIN {X 0,Y 376.359,Z 776.717,A -85,B 0,C 180,E1 -12286.743,E2 -12286.743} C_VEL
LIN {X 0,Y 377.307,Z 782.082,A -85,B 0,C 180,E1 -12289.792,E2 -12289.792} C_VEL
LIN {X 0,Y 378.284,Z 788.033,A -85,B 0,C 180,E1 -12293.025,E2 -12293.025} C_VEL
LIN {X 0,Y 378.226,Z 791.596,A -85,B 0,C 180,E1 -12294.845,E2 -12294.845} C_VEL
LIN {X 0,Y 377.465,Z 799.207,A -85,B 0,C 180,E1 -12298.578,E2 -12298.578} C_VEL
LIN {X 0,Y 376.598,Z 808.088,A -85,B 0,C 180,E1 -12302.792,E2 -12302.792} C_VEL
LIN {X 0,Y 375.949,Z 815.779,A -85,B 0,C 180,E1 -12306.351,E2 -12306.351} C_VEL
LIN {X 0,Y 375.44,Z 824.126,A -85,B 0,C 180,E1 -12310.14,E2 -12310.14} C_VEL
LIN {X 0,Y 378.226,Z 839.224,A -85,B 0,C 180,E1 -12311.101,E2 -12311.101} C_VEL
LIN {X 0,Y 379.501,Z 852.898,A -85,B 0,C 180,E1 -12312.076,E2 -12312.076} C_VEL
LIN {X 0,Y 380.079,Z 861.288,A -85,B 0,C 180,E1 -12312.791,E2 -12312.791} C_VEL
LIN {X 0,Y 378.953,Z 872.897,A -85,B 0,C 180,E1 -12313.848,E2 -12313.848} C_VEL
LIN {X 0,Y 377.851,Z 884.256,A -85,B 0,C 180,E1 -12315.141,E2 -12315.141} C_VEL
LIN {X 0,Y 376.945,Z 894.135,A -85,B 0,C 180,E1 -12316.523,E2 -12316.523} C_VEL
LIN {X 0,Y 376.056,Z 903.474,A -85,B 0,C 180,E1 -12318.137,E2 -12318.137} C_VEL
LIN {X 0,Y 375.344,Z 912.504,A -85,B 0,C 180,E1 -12320.026,E2 -12320.026} C_VEL
LIN {X 0,Y 374.908,Z 919.681,A -85,B 0,C 180,E1 -12321.918,E2 -12321.918} C_VEL
LIN {X 0,Y 374.708,Z 925.013,A -85,B 0,C 180,E1 -12323.76,E2 -12323.76} C_VEL
LIN {X 0,Y 374.662,Z 928.052,A -85,B 0,C 180,E1 -12325.158,E2 -12325.158} C_VEL
LIN {X 0,Y 374.56,Z 930.596,A -85,B 0,C 180,E1 -12326.773,E2 -12326.773} C_VEL
LIN {X 0,Y 374.695,Z 931.77,A -85,B 0,C 180,E1 -12327.85,E2 -12327.85} C_VEL
LIN {X 0,Y 374.67,Z 932.461,A -85,B 0,C 180,E1 -12328.925,E2 -12328.925} C_VEL
LIN {X 0,Y 374.676,Z 932.739,A -85,B 0,C 180,E1 -12330,E2 -12330} C_VEL
LIN {X 0,Y 374.669,Z 932.603,A -85,B 0,C 180,E1 -12331.075,E2 -12331.075} C_VEL
LIN {X 0,Y 374.664,Z 932.042,A -85,B 0,C 180,E1 -12332.15,E2 -12332.15} C_VEL
LIN {X 0,Y 374.559,Z 931.017,A -85,B 0,C 180,E1 -12333.227,E2 -12333.227} C_VEL
LIN {X 0,Y 374.609,Z 929.58,A -85,B 0,C 180,E1 -12334.304,E2 -12334.304} C_VEL
LIN {X 0,Y 374.672,Z 926.015,A -85,B 0,C 180,E1 -12336.189,E2 -12336.189} C_VEL
LIN {X 0,Y 374.895,Z 920.964,A -85,B 0,C 180,E1 -12338.083,E2 -12338.083} C_VEL
LIN {X 0,Y 375.37,Z 914.307,A -85,B 0,C 180,E1 -12339.973,E2 -12339.973} C_VEL
LIN {X 0,Y 375.96,Z 907.13,A -85,B 0,C 180,E1 -12341.593,E2 -12341.593} C_VEL
LIN {X 0,Y 376.883,Z 898.26,A -85,B 0,C 180,E1 -12343.205,E2 -12343.205} C_VEL
LIN {X 0,Y 377.765,Z 889.372,A -85,B 0,C 180,E1 -12344.546,E2 -12344.546} C_VEL
LIN {X 0,Y 378.857,Z 878.646,A -85,B 0,C 180,E1 -12345.88,E2 -12345.88} C_VEL
LIN {X 0,Y 380.208,Z 866.688,A -85,B 0,C 180,E1 -12347.064,E2 -12347.064} C_VEL
LIN {X 0,Y 380.526,Z 860.45,A -85,B 0,C 180,E1 -12347.604,E2 -12347.604} C_VEL
LIN {X 0,Y 379.83,Z 847.312,A -85,B 0,C 180,E1 -12348.647,E2 -12348.647} C_VEL
LIN {X 0,Y 378.38,Z 835.813,A -85,B 0,C 180,E1 -12349.436,E2 -12349.436} C_VEL
LIN {X 0,Y 375.412,Z 822.106,A -85,B 0,C 180,E1 -12350.31,E2 -12350.31} C_VEL
LIN {X 0,Y 375.984,Z 813.527,A -85,B 0,C 180,E1 -12354.282,E2 -12354.282} C_VEL
LIN {X 0,Y 376.62,Z 806.433,A -85,B 0,C 180,E1 -12357.809,E2 -12357.809} C_VEL
LIN {X 0,Y 377.445,Z 799.774,A -85,B 0,C 180,E1 -12361.424,E2 -12361.424} C_VEL
LIN {X 0,Y 378.104,Z 795.667,A -85,B 0,C 180,E1 -12363.892,E2 -12363.892} C_VEL
LIN {X 0,Y 378.547,Z 791.909,A -85,B 0,C 180,E1 -12366.449,E2 -12366.449} C_VEL
LIN {X 0,Y 378.356,Z 788.621,A -85,B 0,C 180,E1 -12369.165,E2 -12369.165} C_VEL
LIN {X 0,Y 377.956,Z 785.909,A -85,B 0,C 180,E1 -12372.022,E2 -12372.022} C_VEL
LIN {X 0,Y 377.592,Z 783.827,A -85,B 0,C 180,E1 -12375.014,E2 -12375.014} C_VEL
LIN {X 0,Y 377.3,Z 782.438,A -85,B 0,C 180,E1 -12378.166,E2 -12378.166} C_VEL
LIN {X 0,Y 377.168,Z 781.782,A -85,B 0,C 180,E1 -12381.501,E2 -12381.501} C_VEL
LIN {X 0,Y 376.931,Z 781.87,A -85,B 0,C 180,E1 -12384.689,E2 -12384.689} C_VEL
LIN {X 0,Y 376.693,Z 782.372,A -85,B 0,C 180,E1 -12387.243,E2 -12387.243} C_VEL
LIN {X 0,Y 376.406,Z 783.152,A -85,B 0,C 180,E1 -12389.726,E2 -12389.726} C_VEL
LIN {X 0,Y 376.037,Z 784.71,A -85,B 0,C 180,E1 -12393.348,E2 -12393.348} C_VEL
LIN {X 0,Y 375.742,Z 786.613,A -85,B 0,C 180,E1 -12396.871,E2 -12396.871} C_VEL
LIN {X 0,Y 375.58,Z 788.46,A -85,B 0,C 180,E1 -12399.863,E2 -12399.863} C_VEL
LIN {X 0,Y 376.566,Z 791.353,A -85,B 0,C 180,E1 -12400.104,E2 -12400.104} C_VEL
LIN {X 0,Y 380.714,Z 803.126,A -85,B 0,C 180,E1 -12401.099,E2 -12401.099} C_VEL
LIN {X 0,Y 382.707,Z 811.229,A -85,B 0,C 180,E1 -12401.808,E2 -12401.808} C_VEL
LIN {X 0,Y 381.847,Z 823.052,A -85,B 0,C 180,E1 -12402.734,E2 -12402.734} C_VEL
LIN {X 0,Y 380.853,Z 833.49,A -85,B 0,C 180,E1 -12403.747,E2 -12403.747} C_VEL
LIN {X 0,Y 379.597,Z 844.893,A -85,B 0,C 180,E1 -12405.114,E2 -12405.114} C_VEL
LIN {X 0,Y 378.564,Z 853.066,A -85,B 0,C 180,E1 -12406.307,E2 -12406.307} C_VEL
LIN {X 0,Y 377.745,Z 860.64,A -85,B 0,C 180,E1 -12407.645,E2 -12407.645} C_VEL
LIN {X 0,Y 376.852,Z 868.12,A -85,B 0,C 180,E1 -12409.251,E2 -12409.251} C_VEL
LIN {X 0,Y 376.13,Z 874.136,A -85,B 0,C 180,E1 -12410.86,E2 -12410.86} C_VEL
LIN {X 0,Y 375.628,Z 879.187,A -85,B 0,C 180,E1 -12412.583,E2 -12412.583} C_VEL
LIN {X 0,Y 375.018,Z 883.596,A -85,B 0,C 180,E1 -12414.622,E2 -12414.622} C_VEL
LIN {X 0,Y 375.063,Z 885.203,A -85,B 0,C 180,E1 -12415.7,E2 -12415.7} C_VEL
LIN {X 0,Y 374.915,Z 886.42,A -85,B 0,C 180,E1 -12416.775,E2 -12416.775} C_VEL
LIN {X 0,Y 374.795,Z 887.241,A -85,B 0,C 180,E1 -12417.85,E2 -12417.85} C_VEL
LIN {X 0,Y 374.719,Z 887.641,A -85,B 0,C 180,E1 -12418.924,E2 -12418.924} C_VEL
LIN {X 0,Y 374.677,Z 887.611,A -85,B 0,C 180,E1 -12419.999,E2 -12419.999} C_VEL
LIN {X 0,Y 374.696,Z 887.185,A -85,B 0,C 180,E1 -12421.074,E2 -12421.074} C_VEL
LIN {X 0,Y 374.769,Z 886.363,A -85,B 0,C 180,E1 -12422.148,E2 -12422.148} C_VEL
LIN {X 0,Y 374.779,Z 885.097,A -85,B 0,C 180,E1 -12423.224,E2 -12423.224} C_VEL
LIN {X 0,Y 374.838,Z 882.405,A -85,B 0,C 180,E1 -12424.839,E2 -12424.839} C_VEL
LIN {X 0,Y 375.124,Z 878.671,A -85,B 0,C 180,E1 -12426.453,E2 -12426.453} C_VEL
LIN {X 0,Y 375.352,Z 873.803,A -85,B 0,C 180,E1 -12428.071,E2 -12428.071} C_VEL
LIN {X 0,Y 375.989,Z 866.509,A -85,B 0,C 180,E1 -12429.955,E2 -12429.955} C_VEL
LIN {X 0,Y 376.628,Z 858.599,A -85,B 0,C 180,E1 -12431.571,E2 -12431.571} C_VEL
LIN {X 0,Y 377.467,Z 848.752,A -85,B 0,C 180,E1 -12433.183,E2 -12433.183} C_VEL
LIN {X 0,Y 378.391,Z 838.62,A -85,B 0,C 180,E1 -12434.52,E2 -12434.52} C_VEL
LIN {X 0,Y 379.107,Z 827.705,A -85,B 0,C 180,E1 -12435.688,E2 -12435.688} C_VEL
LIN {X 0,Y 379.874,Z 816.385,A -85,B 0,C 180,E1 -12436.663,E2 -12436.663} C_VEL
LIN {X 0,Y 380.375,Z 808.826,A -85,B 0,C 180,E1 -12437.194,E2 -12437.194} C_VEL
LIN {X 0,Y 377.803,Z 796.703,A -85,B 0,C 180,E1 -12438.002,E2 -12438.002} C_VEL
LIN {X 0,Y 374.819,Z 783.488,A -85,B 0,C 180,E1 -12438.693,E2 -12438.693} C_VEL
LIN {X 0,Y 374.862,Z 780.233,A -85,B 0,C 180,E1 -12442.021,E2 -12442.021} C_VEL
LIN {X 0,Y 375.019,Z 776.513,A -85,B 0,C 180,E1 -12445.902,E2 -12445.902} C_VEL
LIN {X 0,Y 375.075,Z 774.767,A -85,B 0,C 180,E1 -12447.932,E2 -12447.932} C_VEL
LIN {X 0,Y 375.498,Z 774.71,A -85,B 0,C 180,E1 -12451.603,E2 -12451.603} C_VEL
LIN {X 0,Y 375.819,Z 774.674,A -85,B 0,C 180,E1 -12454.631,E2 -12454.631} C_VEL
LIN {X 0,Y 375.957,Z 774.654,A -85,B 0,C 180,E1 -12458.088,E2 -12458.088} C_VEL
LIN {X 0,Y 375.935,Z 774.659,A -85,B 0,C 180,E1 -12460.866,E2 -12460.866} C_VEL
LIN {X 0,Y 375.924,Z 774.656,A -85,B 0,C 180,E1 -12463.765,E2 -12463.765} C_VEL
LIN {X 0,Y 375.929,Z 774.659,A -85,B 0,C 180,E1 -12466.809,E2 -12466.809} C_VEL
LIN {X 0,Y 375.955,Z 774.654,A -85,B 0,C 180,E1 -12470.536,E2 -12470.536} C_VEL
LIN {X 0,Y 375.956,Z 774.653,A -85,B 0,C 180,E1 -12473.495,E2 -12473.495} C_VEL
LIN {X 0,Y 375.952,Z 774.652,A -85,B 0,C 180,E1 -12475.888,E2 -12475.888} C_VEL
LIN {X 0,Y 375.954,Z 774.653,A -85,B 0,C 180,E1 -12479.686,E2 -12479.686} C_VEL
LIN {X 0,Y 375.926,Z 774.661,A -85,B 0,C 180,E1 -12483.341,E2 -12483.341} C_VEL
LIN {X 0,Y 375.969,Z 774.652,A -85,B 0,C 180,E1 -12486.886,E2 -12486.886} C_VEL
LIN {X 0,Y 375.987,Z 774.647,A -85,B 0,C 180,E1 -12490.339,E2 -12490.339} C_VEL
LIN {X 0,Y 376.017,Z 774.648,A -85,B 0,C 180,E1 -12493.718,E2 -12493.718} C_VEL
LIN {X 0,Y 376.094,Z 774.635,A -85,B 0,C 180,E1 -12497.042,E2 -12497.042} C_VEL
LIN {X 0,Y 376.102,Z 774.634,A -85,B 0,C 180,E1 -12500.318,E2 -12500.318} C_VEL
LIN {X 0,Y 376.183,Z 774.626,A -85,B 0,C 180,E1 -12503.564,E2 -12503.564} C_VEL
LIN {X 0,Y 376.326,Z 774.61,A -85,B 0,C 180,E1 -12507.859,E2 -12507.859} C_VEL
LIN {X 0,Y 376.321,Z 774.611,A -85,B 0,C 180,E1 -12512.141,E2 -12512.141} C_VEL
LIN {X 0,Y 376.182,Z 774.626,A -85,B 0,C 180,E1 -12516.436,E2 -12516.436} C_VEL
LIN {X 0,Y 376.096,Z 774.634,A -85,B 0,C 180,E1 -12519.682,E2 -12519.682} C_VEL
LIN {X 0,Y 376.08,Z 774.636,A -85,B 0,C 180,E1 -12523.658,E2 -12523.658} C_VEL
LIN {X 0,Y 376.023,Z 774.642,A -85,B 0,C 180,E1 -12527.4,E2 -12527.4} C_VEL
LIN {X 0,Y 375.97,Z 774.652,A -85,B 0,C 180,E1 -12530.833,E2 -12530.833} C_VEL
LIN {X 0,Y 375.962,Z 774.653,A -85,B 0,C 180,E1 -12534.284,E2 -12534.284} C_VEL
LIN {X 0,Y 375.925,Z 774.655,A -85,B 0,C 180,E1 -12537.865,E2 -12537.865} C_VEL
LIN {X 0,Y 375.949,Z 774.653,A -85,B 0,C 180,E1 -12541.563,E2 -12541.563} C_VEL
LIN {X 0,Y 375.95,Z 774.654,A -85,B 0,C 180,E1 -12545.416,E2 -12545.416} C_VEL
LIN {X 0,Y 375.937,Z 774.654,A -85,B 0,C 180,E1 -12546.032,E2 -12546.032} C_VEL
LIN {X 0,Y 375.29,Z 774.74,A -85,B 0,C 180,E1 -12546.926,E2 -12546.926} C_VEL
LIN {X 0,Y 372.455,Z 775.09,A -85,B 0,C 180,E1 -12548.381,E2 -12548.381} C_VEL
LIN {X 0,Y 370.031,Z 775.392,A -85,B 0,C 180,E1 -12549.556,E2 -12549.556} C_VEL
LIN {X 0,Y 368.969,Z 775.523,A -85,B 0,C 180,E1 -12550.465,E2 -12550.465} C_VEL
LIN {X 0,Y 368.873,Z 775.531,A -85,B 0,C 180,E1 -12550.774,E2 -12550.774} C_VEL
LIN {X 0,Y 368.877,Z 775.536,A -85,B 0,C 180,E1 -12553.617,E2 -12553.617} C_VEL
LIN {X 0,Y 368.88,Z 775.534,A -85,B 0,C 180,E1 -12556.697,E2 -12556.697} C_VEL
LIN {X 0,Y 368.907,Z 775.533,A -85,B 0,C 180,E1 -12559.644,E2 -12559.644} C_VEL
LIN {X 0,Y 368.867,Z 775.538,A -85,B 0,C 180,E1 -12563.152,E2 -12563.152} C_VEL
LIN {X 0,Y 368.68,Z 775.558,A -85,B 0,C 180,E1 -12566.441,E2 -12566.441} C_VEL
LIN {X 0,Y 368.381,Z 775.598,A -85,B 0,C 180,E1 -12569.15,E2 -12569.15} C_VEL
LIN {X 0,Y 367.952,Z 775.652,A -85,B 0,C 180,E1 -12572.717,E2 -12572.717} C_VEL
LIN {X 0,Y 367.86,Z 775.814,A -85,B 0,C 180,E1 -12573.935,E2 -12573.935} C_VEL
LIN {X 0,Y 367.728,Z 779.574,A -85,B 0,C 180,E1 -12577.529,E2 -12577.529} C_VEL
LIN {X 0,Y 367.742,Z 783.295,A -85,B 0,C 180,E1 -12581.042,E2 -12581.042} C_VEL
LIN {X 0,Y 367.729,Z 783.422,A -85,B 0,C 180,E1 -12581.159,E2 -12581.159} C_VEL
LIN {X 0,Y 370.704,Z 796.861,A -85,B 0,C 180,E1 -12581.859,E2 -12581.859} C_VEL
LIN {X 0,Y 373.295,Z 809.885,A -85,B 0,C 180,E1 -12582.752,E2 -12582.752} C_VEL
LIN {X 0,Y 372.462,Z 822.255,A -85,B 0,C 180,E1 -12583.701,E2 -12583.701} C_VEL
LIN {X 0,Y 371.723,Z 833.405,A -85,B 0,C 180,E1 -12584.797,E2 -12584.797} C_VEL
LIN {X 0,Y 370.84,Z 844.59,A -85,B 0,C 180,E1 -12586.158,E2 -12586.158} C_VEL
LIN {X 0,Y 369.926,Z 854.499,A -85,B 0,C 180,E1 -12587.66,E2 -12587.66} C_VEL
LIN {X 0,Y 369.184,Z 863.286,A -85,B 0,C 180,E1 -12589.305,E2 -12589.305} C_VEL
LIN {X 0,Y 368.566,Z 870.327,A -85,B 0,C 180,E1 -12590.95,E2 -12590.95} C_VEL
LIN {X 0,Y 368.156,Z 876.34,A -85,B 0,C 180,E1 -12592.721,E2 -12592.721} C_VEL
LIN {X 0,Y 367.871,Z 881.035,A -85,B 0,C 180,E1 -12594.52,E2 -12594.52} C_VEL
LIN {X 0,Y 367.698,Z 883.258,A -85,B 0,C 180,E1 -12595.616,E2 -12595.616} C_VEL
LIN {X 0,Y 367.661,Z 885.01,A -85,B 0,C 180,E1 -12596.714,E2 -12596.714} C_VEL
LIN {X 0,Y 367.694,Z 886.353,A -85,B 0,C 180,E1 -12597.81,E2 -12597.81} C_VEL
LIN {X 0,Y 367.62,Z 887.279,A -85,B 0,C 180,E1 -12598.906,E2 -12598.906} C_VEL
LIN {X 0,Y 367.639,Z 887.848,A -85,B 0,C 180,E1 -12601.096,E2 -12601.096} C_VEL
LIN {X 0,Y 367.717,Z 887.54,A -85,B 0,C 180,E1 -12602.192,E2 -12602.192} C_VEL
LIN {X 0,Y 367.856,Z 886.777,A -85,B 0,C 180,E1 -12603.287,E2 -12603.287} C_VEL
LIN {X 0,Y 367.978,Z 885.613,A -85,B 0,C 180,E1 -12604.383,E2 -12604.383} C_VEL
LIN {X 0,Y 368.101,Z 883.083,A -85,B 0,C 180,E1 -12606.029,E2 -12606.029} C_VEL
LIN {X 0,Y 368.578,Z 879.521,A -85,B 0,C 180,E1 -12607.672,E2 -12607.672} C_VEL
LIN {X 0,Y 369.152,Z 874.87,A -85,B 0,C 180,E1 -12609.314,E2 -12609.314} C_VEL
LIN {X 0,Y 369.827,Z 868.997,A -85,B 0,C 180,E1 -12610.956,E2 -12610.956} C_VEL
LIN {X 0,Y 370.811,Z 861.642,A -85,B 0,C 180,E1 -12612.59,E2 -12612.59} C_VEL
LIN {X 0,Y 371.83,Z 852.551,A -85,B 0,C 180,E1 -12614.225,E2 -12614.225} C_VEL
LIN {X 0,Y 373.199,Z 842.59,A -85,B 0,C 180,E1 -12615.659,E2 -12615.659} C_VEL
LIN {X 0,Y 374.324,Z 831.888,A -85,B 0,C 180,E1 -12616.919,E2 -12616.919} C_VEL
LIN {X 0,Y 375.553,Z 820.491,A -85,B 0,C 180,E1 -12617.987,E2 -12617.987} C_VEL
LIN {X 0,Y 376.154,Z 813.628,A -85,B 0,C 180,E1 -12618.52,E2 -12618.52} C_VEL
LIN {X 0,Y 374.316,Z 804.602,A -85,B 0,C 180,E1 -12619.334,E2 -12619.334} C_VEL
LIN {X 0,Y 370.698,Z 793.6,A -85,B 0,C 180,E1 -12620.303,E2 -12620.303} C_VEL
LIN {X 0,Y 368.43,Z 787.729,A -85,B 0,C 180,E1 -12620.82,E2 -12620.82} C_VEL
LIN {X 0,Y 368.537,Z 784.876,A -85,B 0,C 180,E1 -12623.743,E2 -12623.743} C_VEL
LIN {X 0,Y 368.626,Z 781.526,A -85,B 0,C 180,E1 -12627.231,E2 -12627.231} C_VEL
LIN {X 0,Y 368.698,Z 779.119,A -85,B 0,C 180,E1 -12629.711,E2 -12629.711} C_VEL
LIN {X 0,Y 368.691,Z 776.04,A -85,B 0,C 180,E1 -12632.993,E2 -12632.993} C_VEL
LIN {X 0,Y 368.674,Z 775.564,A -85,B 0,C 180,E1 -12633.562,E2 -12633.562} C_VEL
LIN {X 0,Y 368.874,Z 775.538,A -85,B 0,C 180,E1 -12636.85,E2 -12636.85} C_VEL
LIN {X 0,Y 368.913,Z 775.534,A -85,B 0,C 180,E1 -12640.371,E2 -12640.371} C_VEL
LIN {X 0,Y 368.887,Z 775.535,A -85,B 0,C 180,E1 -12643.616,E2 -12643.616} C_VEL
LIN {X 0,Y 368.919,Z 775.651,A -85,B 0,C 180,E1 -12645.323,E2 -12645.323} C_VEL
LIN {X 0,Y 369.856,Z 780.706,A -85,B 0,C 180,E1 -12648.312,E2 -12648.312} C_VEL
LIN {X 0,Y 371.014,Z 787.239,A -85,B 0,C 180,E1 -12652.002,E2 -12652.002} C_VEL
LIN {X 0,Y 371.293,Z 791.12,A -85,B 0,C 180,E1 -12654.071,E2 -12654.071} C_VEL
LIN {X 0,Y 370.794,Z 796.215,A -85,B 0,C 180,E1 -12656.656,E2 -12656.656} C_VEL
LIN {X 0,Y 370.096,Z 802.555,A -85,B 0,C 180,E1 -12659.786,E2 -12659.786} C_VEL
LIN {X 0,Y 369.402,Z 810.068,A -85,B 0,C 180,E1 -12663.406,E2 -12663.406} C_VEL
LIN {X 0,Y 368.766,Z 817.7,A -85,B 0,C 180,E1 -12667.002,E2 -12667.002} C_VEL
LIN {X 0,Y 368.458,Z 823.159,A -85,B 0,C 180,E1 -12669.537,E2 -12669.537} C_VEL
LIN {X 0,Y 371.635,Z 839.73,A -85,B 0,C 180,E1 -12670.652,E2 -12670.652} C_VEL
LIN {X 0,Y 372.801,Z 853.577,A -85,B 0,C 180,E1 -12671.703,E2 -12671.703} C_VEL
LIN {X 0,Y 373.233,Z 863.733,A -85,B 0,C 180,E1 -12672.607,E2 -12672.607} C_VEL
LIN {X 0,Y 371.941,Z 875.924,A -85,B 0,C 180,E1 -12673.817,E2 -12673.817} C_VEL
LIN {X 0,Y 370.797,Z 886.777,A -85,B 0,C 180,E1 -12675.162,E2 -12675.162} C_VEL
LIN {X 0,Y 369.672,Z 897.536,A -85,B 0,C 180,E1 -12676.813,E2 -12676.813} C_VEL
LIN {X 0,Y 368.839,Z 906.143,A -85,B 0,C 180,E1 -12678.459,E2 -12678.459} C_VEL
LIN {X 0,Y 368.225,Z 913.156,A -85,B 0,C 180,E1 -12680.109,E2 -12680.109} C_VEL
LIN {X 0,Y 367.752,Z 920.703,A -85,B 0,C 180,E1 -12682.312,E2 -12682.312} C_VEL
LIN {X 0,Y 367.641,Z 924.649,A -85,B 0,C 180,E1 -12683.757,E2 -12683.757} C_VEL
LIN {X 0,Y 367.541,Z 928.429,A -85,B 0,C 180,E1 -12685.613,E2 -12685.613} C_VEL
LIN {X 0,Y 367.473,Z 930.044,A -85,B 0,C 180,E1 -12686.711,E2 -12686.711} C_VEL
LIN {X 0,Y 367.609,Z 931.249,A -85,B 0,C 180,E1 -12687.809,E2 -12687.809} C_VEL
LIN {X 0,Y 367.603,Z 931.982,A -85,B 0,C 180,E1 -12688.905,E2 -12688.905} C_VEL
LIN {X 0,Y 367.607,Z 932.278,A -85,B 0,C 180,E1 -12690,E2 -12690} C_VEL
LIN {X 0,Y 367.602,Z 932.161,A -85,B 0,C 180,E1 -12691.095,E2 -12691.095} C_VEL
LIN {X 0,Y 367.565,Z 931.63,A -85,B 0,C 180,E1 -12692.192,E2 -12692.192} C_VEL
LIN {X 0,Y 367.471,Z 930.636,A -85,B 0,C 180,E1 -12693.289,E2 -12693.289} C_VEL
LIN {X 0,Y 367.535,Z 929.225,A -85,B 0,C 180,E1 -12694.387,E2 -12694.387} C_VEL
LIN {X 0,Y 367.568,Z 926.068,A -85,B 0,C 180,E1 -12696.139,E2 -12696.139} C_VEL
LIN {X 0,Y 367.728,Z 922.289,A -85,B 0,C 180,E1 -12697.688,E2 -12697.688} C_VEL
LIN {X 0,Y 368.081,Z 917.146,A -85,B 0,C 180,E1 -12699.34,E2 -12699.34} C_VEL
LIN {X 0,Y 368.728,Z 909.578,A -85,B 0,C 180,E1 -12701.266,E2 -12701.266} C_VEL
LIN {X 0,Y 369.613,Z 901.432,A -85,B 0,C 180,E1 -12702.91,E2 -12702.91} C_VEL
LIN {X 0,Y 370.599,Z 892.088,A -85,B 0,C 180,E1 -12704.454,E2 -12704.454} C_VEL
LIN {X 0,Y 371.772,Z 881.262,A -85,B 0,C 180,E1 -12705.909,E2 -12705.909} C_VEL
LIN {X 0,Y 373.321,Z 868.815,A -85,B 0,C 180,E1 -12707.248,E2 -12707.248} C_VEL
LIN {X 0,Y 373.803,Z 861.388,A -85,B 0,C 180,E1 -12707.931,E2 -12707.931} C_VEL
LIN {X 0,Y 373.25,Z 848.763,A -85,B 0,C 180,E1 -12708.988,E2 -12708.988} C_VEL
LIN {X 0,Y 372.064,Z 838.249,A -85,B 0,C 180,E1 -12709.764,E2 -12709.764} C_VEL
LIN {X 0,Y 369.36,Z 825.338,A -85,B 0,C 180,E1 -12710.659,E2 -12710.659} C_VEL
LIN {X 0,Y 368.447,Z 821.484,A -85,B 0,C 180,E1 -12710.903,E2 -12710.903} C_VEL
LIN {X 0,Y 369.034,Z 813.431,A -85,B 0,C 180,E1 -12714.77,E2 -12714.77} C_VEL
LIN {X 0,Y 369.692,Z 806.439,A -85,B 0,C 180,E1 -12718.376,E2 -12718.376} C_VEL
LIN {X 0,Y 370.645,Z 799.922,A -85,B 0,C 180,E1 -12722.068,E2 -12722.068} C_VEL
LIN {X 0,Y 371.262,Z 795.931,A -85,B 0,C 180,E1 -12724.604,E2 -12724.604} C_VEL
LIN {X 0,Y 371.604,Z 792.32,A -85,B 0,C 180,E1 -12727.244,E2 -12727.244} C_VEL
LIN {X 0,Y 371.286,Z 789.212,A -85,B 0,C 180,E1 -12730.059,E2 -12730.059} C_VEL
LIN {X 0,Y 370.891,Z 786.69,A -85,B 0,C 180,E1 -12733.013,E2 -12733.013} C_VEL
LIN {X 0,Y 370.519,Z 784.813,A -85,B 0,C 180,E1 -12736.12,E2 -12736.12} C_VEL
LIN {X 0,Y 370.284,Z 783.643,A -85,B 0,C 180,E1 -12739.394,E2 -12739.394} C_VEL
LIN {X 0,Y 370.232,Z 783.314,A -85,B 0,C 180,E1 -12741.212,E2 -12741.212} C_VEL
LIN {X 0,Y 369.973,Z 783.323,A -85,B 0,C 180,E1 -12744.769,E2 -12744.769} C_VEL
LIN {X 0,Y 369.628,Z 783.908,A -85,B 0,C 180,E1 -12747.832,E2 -12747.832} C_VEL
LIN {X 0,Y 369.261,Z 784.995,A -85,B 0,C 180,E1 -12751.105,E2 -12751.105} C_VEL
LIN {X 0,Y 368.968,Z 786.277,A -85,B 0,C 180,E1 -12754.016,E2 -12754.016} C_VEL
LIN {X 0,Y 368.674,Z 788.192,A -85,B 0,C 180,E1 -12757.587,E2 -12757.587} C_VEL
LIN {X 0,Y 368.59,Z 789.198,A -85,B 0,C 180,E1 -12759.267,E2 -12759.267} C_VEL
LIN {X 0,Y 369.699,Z 792.256,A -85,B 0,C 180,E1 -12759.537,E2 -12759.537} C_VEL
LIN {X 0,Y 373.698,Z 803.01,A -85,B 0,C 180,E1 -12760.508,E2 -12760.508} C_VEL
LIN {X 0,Y 376.29,Z 813.534,A -85,B 0,C 180,E1 -12761.487,E2 -12761.487} C_VEL
LIN {X 0,Y 375.255,Z 825.003,A -85,B 0,C 180,E1 -12762.421,E2 -12762.421} C_VEL
LIN {X 0,Y 373.991,Z 836.696,A -85,B 0,C 180,E1 -12763.627,E2 -12763.627} C_VEL
LIN {X 0,Y 372.722,Z 847.209,A -85,B 0,C 180,E1 -12764.972,E2 -12764.972} C_VEL
LIN {X 0,Y 371.591,Z 855.807,A -85,B 0,C 180,E1 -12766.324,E2 -12766.324} C_VEL
LIN {X 0,Y 370.577,Z 864.305,A -85,B 0,C 180,E1 -12767.958,E2 -12767.958} C_VEL
LIN {X 0,Y 369.69,Z 871.185,A -85,B 0,C 180,E1 -12769.594,E2 -12769.594} C_VEL
LIN {X 0,Y 369.013,Z 876.666,A -85,B 0,C 180,E1 -12771.235,E2 -12771.235} C_VEL
LIN {X 0,Y 368.458,Z 881.312,A -85,B 0,C 180,E1 -12773.04,E2 -12773.04} C_VEL
LIN {X 0,Y 367.974,Z 884.229,A -85,B 0,C 180,E1 -12774.519,E2 -12774.519} C_VEL
LIN {X 0,Y 368.018,Z 885.8,A -85,B 0,C 180,E1 -12775.618,E2 -12775.618} C_VEL
LIN {X 0,Y 367.868,Z 886.987,A -85,B 0,C 180,E1 -12776.713,E2 -12776.713} C_VEL
LIN {X 0,Y 367.735,Z 887.775,A -85,B 0,C 180,E1 -12777.808,E2 -12777.808} C_VEL
LIN {X 0,Y 367.651,Z 888.118,A -85,B 0,C 180,E1 -12778.904,E2 -12778.904} C_VEL
LIN {X 0,Y 367.607,Z 888.055,A -85,B 0,C 180,E1 -12779.999,E2 -12779.999} C_VEL
LIN {X 0,Y 367.629,Z 887.594,A -85,B 0,C 180,E1 -12781.094,E2 -12781.094} C_VEL
LIN {X 0,Y 367.706,Z 886.727,A -85,B 0,C 180,E1 -12782.19,E2 -12782.19} C_VEL
LIN {X 0,Y 367.688,Z 885.411,A -85,B 0,C 180,E1 -12783.286,E2 -12783.286} C_VEL
LIN {X 0,Y 367.782,Z 882.656,A -85,B 0,C 180,E1 -12784.932,E2 -12784.932} C_VEL
LIN {X 0,Y 368.128,Z 877.971,A -85,B 0,C 180,E1 -12786.905,E2 -12786.905} C_VEL
LIN {X 0,Y 368.482,Z 872.017,A -85,B 0,C 180,E1 -12788.775,E2 -12788.775} C_VEL
LIN {X 0,Y 369.05,Z 865.298,A -85,B 0,C 180,E1 -12790.422,E2 -12790.422} C_VEL
LIN {X 0,Y 369.754,Z 856.988,A -85,B 0,C 180,E1 -12792.067,E2 -12792.067} C_VEL
LIN {X 0,Y 370.526,Z 848.546,A -85,B 0,C 180,E1 -12793.434,E2 -12793.434} C_VEL
LIN {X 0,Y 371.419,Z 838.509,A -85,B 0,C 180,E1 -12794.765,E2 -12794.765} C_VEL
LIN {X 0,Y 372.222,Z 827.169,A -85,B 0,C 180,E1 -12795.986,E2 -12795.986} C_VEL
LIN {X 0,Y 373.035,Z 815.646,A -85,B 0,C 180,E1 -12796.978,E2 -12796.978} C_VEL
LIN {X 0,Y 373.458,Z 809.959,A -85,B 0,C 180,E1 -12797.381,E2 -12797.381} C_VEL
LIN {X 0,Y 370.579,Z 796.432,A -85,B 0,C 180,E1 -12798.307,E2 -12798.307} C_VEL
LIN {X 0,Y 367.765,Z 783.835,A -85,B 0,C 180,E1 -12798.993,E2 -12798.993} C_VEL
LIN {X 0,Y 367.79,Z 780.459,A -85,B 0,C 180,E1 -12802.467,E2 -12802.467} C_VEL
LIN {X 0,Y 367.953,Z 776.984,A -85,B 0,C 180,E1 -12806.14,E2 -12806.14} C_VEL
LIN {X 0,Y 367.947,Z 775.918,A -85,B 0,C 180,E1 -12807.283,E2 -12807.283} C_VEL
LIN {X 0,Y 368.191,Z 775.622,A -85,B 0,C 180,E1 -12809.753,E2 -12809.753} C_VEL
LIN {X 0,Y 368.668,Z 775.56,A -85,B 0,C 180,E1 -12813.56,E2 -12813.56} C_VEL
LIN {X 0,Y 368.866,Z 775.538,A -85,B 0,C 180,E1 -12816.848,E2 -12816.848} C_VEL
LIN {X 0,Y 368.906,Z 775.533,A -85,B 0,C 180,E1 -12820.369,E2 -12820.369} C_VEL
LIN {X 0,Y 368.877,Z 775.534,A -85,B 0,C 180,E1 -12823.615,E2 -12823.615} C_VEL
LIN {X 0,Y 368.88,Z 775.537,A -85,B 0,C 180,E1 -12826.695,E2 -12826.695} C_VEL
LIN {X 0,Y 368.905,Z 775.53,A -85,B 0,C 180,E1 -12829.642,E2 -12829.642} C_VEL
LIN {X 0,Y 368.894,Z 775.536,A -85,B 0,C 180,E1 -12833.143,E2 -12833.143} C_VEL
LIN {X 0,Y 368.889,Z 775.533,A -85,B 0,C 180,E1 -12836.461,E2 -12836.461} C_VEL
LIN {X 0,Y 368.922,Z 775.532,A -85,B 0,C 180,E1 -12839.046,E2 -12839.046} C_VEL
LIN {X 0,Y 368.867,Z 775.536,A -85,B 0,C 180,E1 -12842.789,E2 -12842.789} C_VEL
LIN {X 0,Y 368.919,Z 775.528,A -85,B 0,C 180,E1 -12846.118,E2 -12846.118} C_VEL
LIN {X 0,Y 368.927,Z 775.528,A -85,B 0,C 180,E1 -12849.946,E2 -12849.946} C_VEL
LIN {X 0,Y 368.96,Z 775.527,A -85,B 0,C 180,E1 -12853.398,E2 -12853.398} C_VEL
LIN {X 0,Y 369.048,Z 775.511,A -85,B 0,C 180,E1 -12856.79,E2 -12856.79} C_VEL
LIN {X 0,Y 369.052,Z 775.513,A -85,B 0,C 180,E1 -12860.131,E2 -12860.131} C_VEL
LIN {X 0,Y 369.144,Z 775.502,A -85,B 0,C 180,E1 -12863.441,E2 -12863.441} C_VEL
LIN {X 0,Y 369.29,Z 775.486,A -85,B 0,C 180,E1 -12867.819,E2 -12867.819} C_VEL
LIN {X 0,Y 369.284,Z 775.487,A -85,B 0,C 180,E1 -12872.181,E2 -12872.181} C_VEL
LIN {X 0,Y 369.144,Z 775.502,A -85,B 0,C 180,E1 -12876.559,E2 -12876.559} C_VEL
LIN {X 0,Y 369.047,Z 775.514,A -85,B 0,C 180,E1 -12879.869,E2 -12879.869} C_VEL
LIN {X 0,Y 369.028,Z 775.515,A -85,B 0,C 180,E1 -12883.772,E2 -12883.772} C_VEL
LIN {X 0,Y 368.982,Z 775.52,A -85,B 0,C 180,E1 -12887.743,E2 -12887.743} C_VEL
LIN {X 0,Y 368.901,Z 775.531,A -85,B 0,C 180,E1 -12891.221,E2 -12891.221} C_VEL
LIN {X 0,Y 368.916,Z 775.533,A -85,B 0,C 180,E1 -12894.778,E2 -12894.778} C_VEL
LIN {X 0,Y 368.908,Z 775.532,A -85,B 0,C 180,E1 -12898.442,E2 -12898.442} C_VEL
LIN {X 0,Y 368.903,Z 775.534,A -85,B 0,C 180,E1 -12900.988,E2 -12900.988} C_VEL
LIN {X 0,Y 368.929,Z 775.532,A -85,B 0,C 180,E1 -12904.855,E2 -12904.855} C_VEL
LIN {X 0,Y 368.901,Z 775.532,A -85,B 0,C 180,E1 -12908.641,E2 -12908.641} C_VEL
LIN {X 0,Y 368.873,Z 775.531,A -85,B 0,C 180,E1 -12910.774,E2 -12910.774} C_VEL
LIN {X 0,Y 368.167,Z 775.623,A -85,B 0,C 180,E1 -12911.685,E2 -12911.685} C_VEL
LIN {X 0,Y 365.274,Z 775.987,A -85,B 0,C 180,E1 -12913.166,E2 -12913.166} C_VEL
LIN {X 0,Y 362.868,Z 776.282,A -85,B 0,C 180,E1 -12914.365,E2 -12914.365} C_VEL
LIN {X 0,Y 361.872,Z 776.41,A -85,B 0,C 180,E1 -12915.292,E2 -12915.292} C_VEL
LIN {X 0,Y 361.81,Z 776.416,A -85,B 0,C 180,E1 -12915.606,E2 -12915.606} C_VEL
LIN {X 0,Y 361.831,Z 776.416,A -85,B 0,C 180,E1 -12919.246,E2 -12919.246} C_VEL
LIN {X 0,Y 361.858,Z 776.411,A -85,B 0,C 180,E1 -12921.576,E2 -12921.576} C_VEL
LIN {X 0,Y 361.761,Z 776.42,A -85,B 0,C 180,E1 -12924.681,E2 -12924.681} C_VEL
LIN {X 0,Y 361.603,Z 776.441,A -85,B 0,C 180,E1 -12927.032,E2 -12927.032} C_VEL
LIN {X 0,Y 361.115,Z 776.501,A -85,B 0,C 180,E1 -12930.888,E2 -12930.888} C_VEL
LIN {X 0,Y 360.83,Z 776.542,A -85,B 0,C 180,E1 -12933.632,E2 -12933.632} C_VEL
LIN {X 0,Y 360.719,Z 777.202,A -85,B 0,C 180,E1 -12934.621,E2 -12934.621} C_VEL
LIN {X 0,Y 360.647,Z 781.017,A -85,B 0,C 180,E1 -12938.27,E2 -12938.27} C_VEL
LIN {X 0,Y 360.672,Z 783.861,A -85,B 0,C 180,E1 -12940.897,E2 -12940.897} C_VEL
LIN {X 0,Y 363.757,Z 797.966,A -85,B 0,C 180,E1 -12941.646,E2 -12941.646} C_VEL
LIN {X 0,Y 366.298,Z 809.872,A -85,B 0,C 180,E1 -12942.484,E2 -12942.484} C_VEL
LIN {X 0,Y 365.605,Z 821.477,A -85,B 0,C 180,E1 -12943.386,E2 -12943.386} C_VEL
LIN {X 0,Y 364.809,Z 832.879,A -85,B 0,C 180,E1 -12944.502,E2 -12944.502} C_VEL
LIN {X 0,Y 363.927,Z 844.193,A -85,B 0,C 180,E1 -12945.89,E2 -12945.89} C_VEL
LIN {X 0,Y 363.079,Z 852.593,A -85,B 0,C 180,E1 -12947.139,E2 -12947.139} C_VEL
LIN {X 0,Y 362.443,Z 860.423,A -85,B 0,C 180,E1 -12948.537,E2 -12948.537} C_VEL
LIN {X 0,Y 361.736,Z 868.089,A -85,B 0,C 180,E1 -12950.213,E2 -12950.213} C_VEL
LIN {X 0,Y 361.14,Z 875.2,A -85,B 0,C 180,E1 -12952.172,E2 -12952.172} C_VEL
LIN {X 0,Y 360.921,Z 879.913,A -85,B 0,C 180,E1 -12953.853,E2 -12953.853} C_VEL
LIN {X 0,Y 360.632,Z 883.503,A -85,B 0,C 180,E1 -12955.53,E2 -12955.53} C_VEL
LIN {X 0,Y 360.571,Z 885.297,A -85,B 0,C 180,E1 -12956.649,E2 -12956.649} C_VEL
LIN {X 0,Y 360.613,Z 886.68,A -85,B 0,C 180,E1 -12957.767,E2 -12957.767} C_VEL
LIN {X 0,Y 360.555,Z 887.662,A -85,B 0,C 180,E1 -12958.884,E2 -12958.884} C_VEL
LIN {X 0,Y 360.521,Z 888.187,A -85,B 0,C 180,E1 -12960.001,E2 -12960.001} C_VEL
LIN {X 0,Y 360.574,Z 888.308,A -85,B 0,C 180,E1 -12961.118,E2 -12961.118} C_VEL
LIN {X 0,Y 360.66,Z 888.035,A -85,B 0,C 180,E1 -12962.235,E2 -12962.235} C_VEL
LIN {X 0,Y 360.81,Z 887.328,A -85,B 0,C 180,E1 -12963.351,E2 -12963.351} C_VEL
LIN {X 0,Y 360.917,Z 886.205,A -85,B 0,C 180,E1 -12964.468,E2 -12964.468} C_VEL
LIN {X 0,Y 360.902,Z 884.7,A -85,B 0,C 180,E1 -12965.589,E2 -12965.589} C_VEL
LIN {X 0,Y 361.533,Z 881.011,A -85,B 0,C 180,E1 -12967.513,E2 -12967.513} C_VEL
LIN {X 0,Y 362.211,Z 875.693,A -85,B 0,C 180,E1 -12969.494,E2 -12969.494} C_VEL
LIN {X 0,Y 362.921,Z 869.892,A -85,B 0,C 180,E1 -12971.167,E2 -12971.167} C_VEL
LIN {X 0,Y 363.966,Z 862.718,A -85,B 0,C 180,E1 -12972.831,E2 -12972.831} C_VEL
LIN {X 0,Y 365.064,Z 853.82,A -85,B 0,C 180,E1 -12974.494,E2 -12974.494} C_VEL
LIN {X 0,Y 366.524,Z 843.85,A -85,B 0,C 180,E1 -12975.982,E2 -12975.982} C_VEL
LIN {X 0,Y 367.837,Z 832.324,A -85,B 0,C 180,E1 -12977.37,E2 -12977.37} C_VEL
LIN {X 0,Y 369.164,Z 821.055,A -85,B 0,C 180,E1 -12978.452,E2 -12978.452} C_VEL
LIN {X 0,Y 369.654,Z 814.273,A -85,B 0,C 180,E1 -12979.01,E2 -12979.01} C_VEL
LIN {X 0,Y 367.433,Z 804.566,A -85,B 0,C 180,E1 -12979.938,E2 -12979.938} C_VEL
LIN {X 0,Y 363.67,Z 794.02,A -85,B 0,C 180,E1 -12980.952,E2 -12980.952} C_VEL
LIN {X 0,Y 361.451,Z 788.379,A -85,B 0,C 180,E1 -12981.48,E2 -12981.48} C_VEL
LIN {X 0,Y 361.562,Z 785.878,A -85,B 0,C 180,E1 -12984.093,E2 -12984.093} C_VEL
LIN {X 0,Y 361.678,Z 782.419,A -85,B 0,C 180,E1 -12987.799,E2 -12987.799} C_VEL
LIN {X 0,Y 361.786,Z 779.229,A -85,B 0,C 180,E1 -12991.269,E2 -12991.269} C_VEL
LIN {X 0,Y 361.709,Z 776.432,A -85,B 0,C 180,E1 -12994.466,E2 -12994.466} C_VEL
LIN {X 0,Y 361.839,Z 776.414,A -85,B 0,C 180,E1 -12997.217,E2 -12997.217} C_VEL
LIN {X 0,Y 361.857,Z 776.412,A -85,B 0,C 180,E1 -12999.862,E2 -12999.862} C_VEL
LIN {X 0,Y 361.84,Z 776.414,A -85,B 0,C 180,E1 -13002.829,E2 -13002.829} C_VEL
LIN {X 0,Y 361.857,Z 776.495,A -85,B 0,C 180,E1 -13005.028,E2 -13005.028} C_VEL
LIN {X 0,Y 362.832,Z 781.631,A -85,B 0,C 180,E1 -13008.141,E2 -13008.141} C_VEL
LIN {X 0,Y 363.959,Z 788.045,A -85,B 0,C 180,E1 -13011.836,E2 -13011.836} C_VEL
LIN {X 0,Y 364.257,Z 792.263,A -85,B 0,C 180,E1 -13014.132,E2 -13014.132} C_VEL
LIN {X 0,Y 363.749,Z 797.218,A -85,B 0,C 180,E1 -13016.695,E2 -13016.695} C_VEL
LIN {X 0,Y 363.044,Z 803.341,A -85,B 0,C 180,E1 -13019.78,E2 -13019.78} C_VEL
LIN {X 0,Y 362.289,Z 810.909,A -85,B 0,C 180,E1 -13023.501,E2 -13023.501} C_VEL
LIN {X 0,Y 361.648,Z 818.432,A -85,B 0,C 180,E1 -13027.128,E2 -13027.128} C_VEL
LIN {X 0,Y 361.428,Z 822.102,A -85,B 0,C 180,E1 -13028.877,E2 -13028.877} C_VEL
LIN {X 0,Y 362.233,Z 825.793,A -85,B 0,C 180,E1 -13029.121,E2 -13029.121} C_VEL
LIN {X 0,Y 365.005,Z 840.079,A -85,B 0,C 180,E1 -13030.162,E2 -13030.162} C_VEL
LIN {X 0,Y 366.174,Z 854.52,A -85,B 0,C 180,E1 -13031.324,E2 -13031.324} C_VEL
LIN {X 0,Y 366.524,Z 864.639,A -85,B 0,C 180,E1 -13032.278,E2 -13032.278} C_VEL
LIN {X 0,Y 365.171,Z 876.473,A -85,B 0,C 180,E1 -13033.508,E2 -13033.508} C_VEL
LIN {X 0,Y 363.869,Z 887.683,A -85,B 0,C 180,E1 -13034.96,E2 -13034.96} C_VEL
LIN {X 0,Y 362.76,Z 897.666,A -85,B 0,C 180,E1 -13036.557,E2 -13036.557} C_VEL
LIN {X 0,Y 361.864,Z 906.101,A -85,B 0,C 180,E1 -13038.233,E2 -13038.233} C_VEL
LIN {X 0,Y 361.198,Z 913.03,A -85,B 0,C 180,E1 -13039.914,E2 -13039.914} C_VEL
LIN {X 0,Y 360.802,Z 918.613,A -85,B 0,C 180,E1 -13041.599,E2 -13041.599} C_VEL
LIN {X 0,Y 360.554,Z 924.341,A -85,B 0,C 180,E1 -13043.78,E2 -13043.78} C_VEL
LIN {X 0,Y 360.48,Z 927.84,A -85,B 0,C 180,E1 -13045.527,E2 -13045.527} C_VEL
LIN {X 0,Y 360.39,Z 929.476,A -85,B 0,C 180,E1 -13046.646,E2 -13046.646} C_VEL
LIN {X 0,Y 360.526,Z 930.705,A -85,B 0,C 180,E1 -13047.766,E2 -13047.766} C_VEL
LIN {X 0,Y 360.538,Z 931.489,A -85,B 0,C 180,E1 -13048.883,E2 -13048.883} C_VEL
LIN {X 0,Y 360.539,Z 931.81,A -85,B 0,C 180,E1 -13050,E2 -13050} C_VEL
LIN {X 0,Y 360.536,Z 931.72,A -85,B 0,C 180,E1 -13051.117,E2 -13051.117} C_VEL
LIN {X 0,Y 360.467,Z 931.211,A -85,B 0,C 180,E1 -13052.235,E2 -13052.235} C_VEL
LIN {X 0,Y 360.387,Z 930.267,A -85,B 0,C 180,E1 -13053.354,E2 -13053.354} C_VEL
LIN {X 0,Y 360.441,Z 928.877,A -85,B 0,C 180,E1 -13054.473,E2 -13054.473} C_VEL
LIN {X 0,Y 360.481,Z 926.071,A -85,B 0,C 180,E1 -13056.112,E2 -13056.112} C_VEL
LIN {X 0,Y 360.677,Z 922.039,A -85,B 0,C 180,E1 -13057.84,E2 -13057.84} C_VEL
LIN {X 0,Y 361.033,Z 916.986,A -85,B 0,C 180,E1 -13059.524,E2 -13059.524} C_VEL
LIN {X 0,Y 361.75,Z 909.511,A -85,B 0,C 180,E1 -13061.486,E2 -13061.486} C_VEL
LIN {X 0,Y 362.683,Z 901.476,A -85,B 0,C 180,E1 -13063.161,E2 -13063.161} C_VEL
LIN {X 0,Y 363.795,Z 891.705,A -85,B 0,C 180,E1 -13064.822,E2 -13064.822} C_VEL
LIN {X 0,Y 364.981,Z 881.751,A -85,B 0,C 180,E1 -13066.213,E2 -13066.213} C_VEL
LIN {X 0,Y 366.397,Z 870.894,A -85,B 0,C 180,E1 -13067.44,E2 -13067.44} C_VEL
LIN {X 0,Y 367.156,Z 863.844,A -85,B 0,C 180,E1 -13068.123,E2 -13068.123} C_VEL
LIN {X 0,Y 366.719,Z 850.646,A -85,B 0,C 180,E1 -13069.315,E2 -13069.315} C_VEL
LIN {X 0,Y 365.736,Z 840.411,A -85,B 0,C 180,E1 -13070.127,E2 -13070.127} C_VEL
LIN {X 0,Y 362.982,Z 827.022,A -85,B 0,C 180,E1 -13071.132,E2 -13071.132} C_VEL
LIN {X 0,Y 361.436,Z 820.801,A -85,B 0,C 180,E1 -13071.582,E2 -13071.582} C_VEL
LIN {X 0,Y 362.067,Z 813.354,A -85,B 0,C 180,E1 -13075.28,E2 -13075.28} C_VEL
LIN {X 0,Y 362.814,Z 806.477,A -85,B 0,C 180,E1 -13078.965,E2 -13078.965} C_VEL
LIN {X 0,Y 363.815,Z 800.111,A -85,B 0,C 180,E1 -13082.744,E2 -13082.744} C_VEL
LIN {X 0,Y 364.433,Z 796.235,A -85,B 0,C 180,E1 -13085.348,E2 -13085.348} C_VEL
LIN {X 0,Y 364.578,Z 792.786,A -85,B 0,C 180,E1 -13088.088,E2 -13088.088} C_VEL
LIN {X 0,Y 364.215,Z 789.864,A -85,B 0,C 180,E1 -13091.001,E2 -13091.001} C_VEL
LIN {X 0,Y 363.842,Z 787.528,A -85,B 0,C 180,E1 -13094.058,E2 -13094.058} C_VEL
LIN {X 0,Y 363.514,Z 785.803,A -85,B 0,C 180,E1 -13097.415,E2 -13097.415} C_VEL
LIN {X 0,Y 363.301,Z 784.912,A -85,B 0,C 180,E1 -13100.696,E2 -13100.696} C_VEL
LIN {X 0,Y 363.15,Z 784.704,A -85,B 0,C 180,E1 -13103.133,E2 -13103.133} C_VEL
LIN {X 0,Y 362.883,Z 784.978,A -85,B 0,C 180,E1 -13106.387,E2 -13106.387} C_VEL
LIN {X 0,Y 362.43,Z 785.83,A -85,B 0,C 180,E1 -13109.722,E2 -13109.722} C_VEL
LIN {X 0,Y 362.05,Z 787.282,A -85,B 0,C 180,E1 -13113.482,E2 -13113.482} C_VEL
LIN {X 0,Y 361.703,Z 789.111,A -85,B 0,C 180,E1 -13117.131,E2 -13117.131} C_VEL
LIN {X 0,Y 361.605,Z 789.952,A -85,B 0,C 180,E1 -13118.6,E2 -13118.6} C_VEL
LIN {X 0,Y 362.876,Z 793.168,A -85,B 0,C 180,E1 -13118.91,E2 -13118.91} C_VEL
LIN {X 0,Y 366.722,Z 803.147,A -85,B 0,C 180,E1 -13119.894,E2 -13119.894} C_VEL
LIN {X 0,Y 369.466,Z 812.981,A -85,B 0,C 180,E1 -13120.862,E2 -13120.862} C_VEL
LIN {X 0,Y 369.841,Z 816.088,A -85,B 0,C 180,E1 -13121.152,E2 -13121.152} C_VEL
LIN {X 0,Y 368.505,Z 828.368,A -85,B 0,C 180,E1 -13122.232,E2 -13122.232} C_VEL
LIN {X 0,Y 367.213,Z 839.509,A -85,B 0,C 180,E1 -13123.466,E2 -13123.466} C_VEL
LIN {X 0,Y 365.761,Z 850.417,A -85,B 0,C 180,E1 -13124.965,E2 -13124.965} C_VEL
LIN {X 0,Y 364.619,Z 858.574,A -85,B 0,C 180,E1 -13126.341,E2 -13126.341} C_VEL
LIN {X 0,Y 363.545,Z 866.568,A -85,B 0,C 180,E1 -13128.004,E2 -13128.004} C_VEL
LIN {X 0,Y 362.515,Z 874.022,A -85,B 0,C 180,E1 -13129.95,E2 -13129.95} C_VEL
LIN {X 0,Y 361.87,Z 879.026,A -85,B 0,C 180,E1 -13131.623,E2 -13131.623} C_VEL
LIN {X 0,Y 361.305,Z 882.896,A -85,B 0,C 180,E1 -13133.297,E2 -13133.297} C_VEL
LIN {X 0,Y 360.934,Z 884.889,A -85,B 0,C 180,E1 -13134.412,E2 -13134.412} C_VEL
LIN {X 0,Y 360.975,Z 886.412,A -85,B 0,C 180,E1 -13135.532,E2 -13135.532} C_VEL
LIN {X 0,Y 360.822,Z 887.556,A -85,B 0,C 180,E1 -13136.649,E2 -13136.649} C_VEL
LIN {X 0,Y 360.677,Z 888.297,A -85,B 0,C 180,E1 -13137.765,E2 -13137.765} C_VEL
LIN {X 0,Y 360.585,Z 888.594,A -85,B 0,C 180,E1 -13138.882,E2 -13138.882} C_VEL
LIN {X 0,Y 360.54,Z 888.495,A -85,B 0,C 180,E1 -13139.999,E2 -13139.999} C_VEL
LIN {X 0,Y 360.564,Z 887.998,A -85,B 0,C 180,E1 -13141.116,E2 -13141.116} C_VEL
LIN {X 0,Y 360.625,Z 887.07,A -85,B 0,C 180,E1 -13142.233,E2 -13142.233} C_VEL
LIN {X 0,Y 360.598,Z 885.714,A -85,B 0,C 180,E1 -13143.351,E2 -13143.351} C_VEL
LIN {X 0,Y 360.73,Z 882.879,A -85,B 0,C 180,E1 -13145.029,E2 -13145.029} C_VEL
LIN {X 0,Y 361.059,Z 878.17,A -85,B 0,C 180,E1 -13147.015,E2 -13147.015} C_VEL
LIN {X 0,Y 361.455,Z 872.023,A -85,B 0,C 180,E1 -13148.947,E2 -13148.947} C_VEL
LIN {X 0,Y 362.054,Z 865.216,A -85,B 0,C 180,E1 -13150.625,E2 -13150.625} C_VEL
LIN {X 0,Y 362.776,Z 856.809,A -85,B 0,C 180,E1 -13152.303,E2 -13152.303} C_VEL
LIN {X 0,Y 363.604,Z 848.241,A -85,B 0,C 180,E1 -13153.695,E2 -13153.695} C_VEL
LIN {X 0,Y 364.572,Z 837.069,A -85,B 0,C 180,E1 -13155.169,E2 -13155.169} C_VEL
LIN {X 0,Y 365.395,Z 826.139,A -85,B 0,C 180,E1 -13156.336,E2 -13156.336} C_VEL
LIN {X 0,Y 366.339,Z 812.888,A -85,B 0,C 180,E1 -13157.442,E2 -13157.442} C_VEL
LIN {X 0,Y 366.362,Z 809.941,A -85,B 0,C 180,E1 -13157.657,E2 -13157.657} C_VEL
LIN {X 0,Y 363.368,Z 796.195,A -85,B 0,C 180,E1 -13158.608,E2 -13158.608} C_VEL
LIN {X 0,Y 360.693,Z 784.223,A -85,B 0,C 180,E1 -13159.25,E2 -13159.25} C_VEL
LIN {X 0,Y 360.759,Z 780.688,A -85,B 0,C 180,E1 -13162.93,E2 -13162.93} C_VEL
LIN {X 0,Y 360.885,Z 777.243,A -85,B 0,C 180,E1 -13166.608,E2 -13166.608} C_VEL
LIN {X 0,Y 360.929,Z 776.528,A -85,B 0,C 180,E1 -13167.859,E2 -13167.859} C_VEL
LIN {X 0,Y 361.38,Z 776.469,A -85,B 0,C 180,E1 -13171.673,E2 -13171.673} C_VEL
LIN {X 0,Y 361.688,Z 776.434,A -85,B 0,C 180,E1 -13174.297,E2 -13174.297} C_VEL
LIN {X 0,Y 361.831,Z 776.412,A -85,B 0,C 180,E1 -13177.216,E2 -13177.216} C_VEL
LIN {X 0,Y 361.85,Z 776.409,A -85,B 0,C 180,E1 -13179.86,E2 -13179.86} C_VEL
LIN {X 0,Y 361.831,Z 776.416,A -85,B 0,C 180,E1 -13182.828,E2 -13182.828} C_VEL
LIN {X 0,Y 361.812,Z 776.413,A -85,B 0,C 180,E1 -13185.945,E2 -13185.945} C_VEL
LIN {X 0,Y 361.829,Z 776.414,A -85,B 0,C 180,E1 -13189.244,E2 -13189.244} C_VEL
LIN {X 0,Y 361.856,Z 776.411,A -85,B 0,C 180,E1 -13192.776,E2 -13192.776} C_VEL
LIN {X 0,Y 361.847,Z 776.41,A -85,B 0,C 180,E1 -13195.719,E2 -13195.719} C_VEL
LIN {X 0,Y 361.857,Z 776.409,A -85,B 0,C 180,E1 -13199.67,E2 -13199.67} C_VEL
LIN {X 0,Y 361.865,Z 776.411,A -85,B 0,C 180,E1 -13203.468,E2 -13203.468} C_VEL
LIN {X 0,Y 361.87,Z 776.409,A -85,B 0,C 180,E1 -13207.143,E2 -13207.143} C_VEL
LIN {X 0,Y 361.877,Z 776.405,A -85,B 0,C 180,E1 -13210.722,E2 -13210.722} C_VEL
LIN {X 0,Y 361.934,Z 776.398,A -85,B 0,C 180,E1 -13214.226,E2 -13214.226} C_VEL
LIN {X 0,Y 361.99,Z 776.391,A -85,B 0,C 180,E1 -13216.527,E2 -13216.527} C_VEL
LIN {X 0,Y 361.989,Z 776.395,A -85,B 0,C 180,E1 -13219.937,E2 -13219.937} C_VEL
LIN {X 0,Y 362.108,Z 776.377,A -85,B 0,C 180,E1 -13223.313,E2 -13223.313} C_VEL
LIN {X 0,Y 362.253,Z 776.362,A -85,B 0,C 180,E1 -13227.776,E2 -13227.776} C_VEL
LIN {X 0,Y 362.163,Z 776.368,A -85,B 0,C 180,E1 -13231.112,E2 -13231.112} C_VEL
LIN {X 0,Y 362.246,Z 776.363,A -85,B 0,C 180,E1 -13232.224,E2 -13232.224} C_VEL
LIN {X 0,Y 362.108,Z 776.377,A -85,B 0,C 180,E1 -13236.687,E2 -13236.687} C_VEL
LIN {X 0,Y 361.984,Z 776.395,A -85,B 0,C 180,E1 -13240.063,E2 -13240.063} C_VEL
LIN {X 0,Y 361.989,Z 776.392,A -85,B 0,C 180,E1 -13243.899,E2 -13243.899} C_VEL
LIN {X 0,Y 361.919,Z 776.401,A -85,B 0,C 180,E1 -13246.935,E2 -13246.935} C_VEL
LIN {X 0,Y 361.878,Z 776.41,A -85,B 0,C 180,E1 -13250.462,E2 -13250.462} C_VEL
LIN {X 0,Y 361.885,Z 776.405,A -85,B 0,C 180,E1 -13254.113,E2 -13254.113} C_VEL
LIN {X 0,Y 361.837,Z 776.41,A -85,B 0,C 180,E1 -13257.785,E2 -13257.785} C_VEL
LIN {X 0,Y 361.839,Z 776.412,A -85,B 0,C 180,E1 -13261.286,E2 -13261.286} C_VEL
LIN {X 0,Y 361.847,Z 776.409,A -85,B 0,C 180,E1 -13264.281,E2 -13264.281} C_VEL
LIN {X 0,Y 361.857,Z 776.411,A -85,B 0,C 180,E1 -13267.224,E2 -13267.224} C_VEL
LIN {X 0,Y 361.829,Z 776.414,A -85,B 0,C 180,E1 -13270.766,E2 -13270.766} C_VEL
LIN {X 0,Y 361.811,Z 776.413,A -85,B 0,C 180,E1 -13274.37,E2 -13274.37} C_VEL
LIN {X 0,Y 361.81,Z 776.416,A -85,B 0,C 180,E1 -13275.606,E2 -13275.606} C_VEL
LIN {X 0,Y 361.179,Z 776.5,A -85,B 0,C 180,E1 -13276.536,E2 -13276.536} C_VEL
LIN {X 0,Y 358.301,Z 776.856,A -85,B 0,C 180,E1 -13278.047,E2 -13278.047} C_VEL
LIN {X 0,Y 355.869,Z 777.159,A -85,B 0,C 180,E1 -13279.271,E2 -13279.271} C_VEL
LIN {X 0,Y 354.871,Z 777.278,A -85,B 0,C 180,E1 -13280.218,E2 -13280.218} C_VEL
LIN {X 0,Y 354.816,Z 777.285,A -85,B 0,C 180,E1 -13280.538,E2 -13280.538} C_VEL
LIN {X 0,Y 354.742,Z 777.298,A -85,B 0,C 180,E1 -13283.536,E2 -13283.536} C_VEL
LIN {X 0,Y 354.621,Z 777.31,A -85,B 0,C 180,E1 -13286.343,E2 -13286.343} C_VEL
LIN {X 0,Y 354.306,Z 777.349,A -85,B 0,C 180,E1 -13288.955,E2 -13288.955} C_VEL
LIN {X 0,Y 353.989,Z 777.393,A -85,B 0,C 180,E1 -13291.545,E2 -13291.545} C_VEL
LIN {X 0,Y 353.701,Z 777.43,A -85,B 0,C 180,E1 -13294.08,E2 -13294.08} C_VEL
LIN {X 0,Y 353.578,Z 781.176,A -85,B 0,C 180,E1 -13297.813,E2 -13297.813} C_VEL
LIN {X 0,Y 353.611,Z 784.129,A -85,B 0,C 180,E1 -13300.613,E2 -13300.613} C_VEL
LIN {X 0,Y 356.57,Z 797.917,A -85,B 0,C 180,E1 -13301.363,E2 -13301.363} C_VEL
LIN {X 0,Y 359.279,Z 810.749,A -85,B 0,C 180,E1 -13302.289,E2 -13302.289} C_VEL
LIN {X 0,Y 358.621,Z 822.125,A -85,B 0,C 180,E1 -13303.2,E2 -13303.2} C_VEL
LIN {X 0,Y 357.831,Z 833.205,A -85,B 0,C 180,E1 -13304.308,E2 -13304.308} C_VEL
LIN {X 0,Y 356.902,Z 844.742,A -85,B 0,C 180,E1 -13305.752,E2 -13305.752} C_VEL
LIN {X 0,Y 355.971,Z 853.981,A -85,B 0,C 180,E1 -13307.168,E2 -13307.168} C_VEL
LIN {X 0,Y 355.166,Z 862.985,A -85,B 0,C 180,E1 -13308.877,E2 -13308.877} C_VEL
LIN {X 0,Y 354.495,Z 870.292,A -85,B 0,C 180,E1 -13310.588,E2 -13310.588} C_VEL
LIN {X 0,Y 354.089,Z 875.239,A -85,B 0,C 180,E1 -13312.015,E2 -13312.015} C_VEL
LIN {X 0,Y 353.86,Z 879.658,A -85,B 0,C 180,E1 -13313.577,E2 -13313.577} C_VEL
LIN {X 0,Y 353.57,Z 883.731,A -85,B 0,C 180,E1 -13315.441,E2 -13315.441} C_VEL
LIN {X 0,Y 353.482,Z 885.585,A -85,B 0,C 180,E1 -13316.582,E2 -13316.582} C_VEL
LIN {X 0,Y 353.534,Z 887.005,A -85,B 0,C 180,E1 -13317.723,E2 -13317.723} C_VEL
LIN {X 0,Y 353.492,Z 888.026,A -85,B 0,C 180,E1 -13318.862,E2 -13318.862} C_VEL
LIN {X 0,Y 353.456,Z 888.614,A -85,B 0,C 180,E1 -13320.001,E2 -13320.001} C_VEL
LIN {X 0,Y 353.51,Z 888.773,A -85,B 0,C 180,E1 -13321.14,E2 -13321.14} C_VEL
LIN {X 0,Y 353.605,Z 888.54,A -85,B 0,C 180,E1 -13322.279,E2 -13322.279} C_VEL
LIN {X 0,Y 353.764,Z 887.905,A -85,B 0,C 180,E1 -13323.418,E2 -13323.418} C_VEL
LIN {X 0,Y 353.86,Z 886.823,A -85,B 0,C 180,E1 -13324.558,E2 -13324.558} C_VEL
LIN {X 0,Y 353.868,Z 885.353,A -85,B 0,C 180,E1 -13325.7,E2 -13325.7} C_VEL
LIN {X 0,Y 354.506,Z 881.904,A -85,B 0,C 180,E1 -13327.589,E2 -13327.589} C_VEL
LIN {X 0,Y 355.037,Z 878.173,A -85,B 0,C 180,E1 -13329.113,E2 -13329.113} C_VEL
LIN {X 0,Y 355.916,Z 871.933,A -85,B 0,C 180,E1 -13331.101,E2 -13331.101} C_VEL
LIN {X 0,Y 356.925,Z 865.107,A -85,B 0,C 180,E1 -13332.799,E2 -13332.799} C_VEL
LIN {X 0,Y 358.17,Z 856.693,A -85,B 0,C 180,E1 -13334.489,E2 -13334.489} C_VEL
LIN {X 0,Y 359.64,Z 846.623,A -85,B 0,C 180,E1 -13336.109,E2 -13336.109} C_VEL
LIN {X 0,Y 361.104,Z 835.464,A -85,B 0,C 180,E1 -13337.558,E2 -13337.558} C_VEL
LIN {X 0,Y 362.619,Z 823.328,A -85,B 0,C 180,E1 -13338.798,E2 -13338.798} C_VEL
LIN {X 0,Y 363.295,Z 816.172,A -85,B 0,C 180,E1 -13339.408,E2 -13339.408} C_VEL
LIN {X 0,Y 361.32,Z 807.219,A -85,B 0,C 180,E1 -13340.332,E2 -13340.332} C_VEL
LIN {X 0,Y 357.308,Z 795.784,A -85,B 0,C 180,E1 -13341.502,E2 -13341.502} C_VEL
LIN {X 0,Y 354.548,Z 789.441,A -85,B 0,C 180,E1 -13342.164,E2 -13342.164} C_VEL
LIN {X 0,Y 354.479,Z 789.053,A -85,B 0,C 180,E1 -13342.207,E2 -13342.207} C_VEL
LIN {X 0,Y 354.597,Z 786.839,A -85,B 0,C 180,E1 -13344.597,E2 -13344.597} C_VEL
LIN {X 0,Y 354.752,Z 783.377,A -85,B 0,C 180,E1 -13348.391,E2 -13348.391} C_VEL
LIN {X 0,Y 354.877,Z 780.551,A -85,B 0,C 180,E1 -13351.616,E2 -13351.616} C_VEL
LIN {X 0,Y 354.86,Z 778.75,A -85,B 0,C 180,E1 -13353.715,E2 -13353.715} C_VEL
LIN {X 0,Y 354.736,Z 777.299,A -85,B 0,C 180,E1 -13355.68,E2 -13355.68} C_VEL
LIN {X 0,Y 354.829,Z 777.286,A -85,B 0,C 180,E1 -13359.424,E2 -13359.424} C_VEL
LIN {X 0,Y 354.792,Z 777.293,A -85,B 0,C 180,E1 -13362.868,E2 -13362.868} C_VEL
LIN {X 0,Y 354.823,Z 777.448,A -85,B 0,C 180,E1 -13364.811,E2 -13364.811} C_VEL
LIN {X 0,Y 355.743,Z 782.271,A -85,B 0,C 180,E1 -13367.801,E2 -13367.801} C_VEL
LIN {X 0,Y 356.673,Z 787.52,A -85,B 0,C 180,E1 -13370.91,E2 -13370.91} C_VEL
LIN {X 0,Y 357.236,Z 791.423,A -85,B 0,C 180,E1 -13373.128,E2 -13373.128} C_VEL
LIN {X 0,Y 356.934,Z 796.396,A -85,B 0,C 180,E1 -13375.791,E2 -13375.791} C_VEL
LIN {X 0,Y 355.979,Z 804.104,A -85,B 0,C 180,E1 -13379.773,E2 -13379.773} C_VEL
LIN {X 0,Y 355.204,Z 811.641,A -85,B 0,C 180,E1 -13383.565,E2 -13383.565} C_VEL
LIN {X 0,Y 354.558,Z 819.132,A -85,B 0,C 180,E1 -13387.261,E2 -13387.261} C_VEL
LIN {X 0,Y 354.449,Z 821.131,A -85,B 0,C 180,E1 -13388.154,E2 -13388.154} C_VEL
LIN {X 0,Y 355.261,Z 824.72,A -85,B 0,C 180,E1 -13388.403,E2 -13388.403} C_VEL
LIN {X 0,Y 357.702,Z 836.139,A -85,B 0,C 180,E1 -13389.289,E2 -13389.289} C_VEL
LIN {X 0,Y 359.043,Z 845.936,A -85,B 0,C 180,E1 -13390.087,E2 -13390.087} C_VEL
LIN {X 0,Y 359.695,Z 858.497,A -85,B 0,C 180,E1 -13391.211,E2 -13391.211} C_VEL
LIN {X 0,Y 359.847,Z 865.65,A -85,B 0,C 180,E1 -13391.938,E2 -13391.938} C_VEL
LIN {X 0,Y 358.565,Z 876.001,A -85,B 0,C 180,E1 -13393.049,E2 -13393.049} C_VEL
LIN {X 0,Y 357.135,Z 887.248,A -85,B 0,C 180,E1 -13394.545,E2 -13394.545} C_VEL
LIN {X 0,Y 356.035,Z 896.253,A -85,B 0,C 180,E1 -13396.007,E2 -13396.007} C_VEL
LIN {X 0,Y 355.017,Z 904.884,A -85,B 0,C 180,E1 -13397.713,E2 -13397.713} C_VEL
LIN {X 0,Y 354.185,Z 912.961,A -85,B 0,C 180,E1 -13399.713,E2 -13399.713} C_VEL
LIN {X 0,Y 353.732,Z 918.437,A -85,B 0,C 180,E1 -13401.43,E2 -13401.43} C_VEL
LIN {X 0,Y 353.507,Z 922.733,A -85,B 0,C 180,E1 -13403.149,E2 -13403.149} C_VEL
LIN {X 0,Y 353.421,Z 927.216,A -85,B 0,C 180,E1 -13405.438,E2 -13405.438} C_VEL
LIN {X 0,Y 353.31,Z 928.885,A -85,B 0,C 180,E1 -13406.579,E2 -13406.579} C_VEL
LIN {X 0,Y 353.445,Z 930.145,A -85,B 0,C 180,E1 -13407.721,E2 -13407.721} C_VEL
LIN {X 0,Y 353.474,Z 930.976,A -85,B 0,C 180,E1 -13408.861,E2 -13408.861} C_VEL
LIN {X 0,Y 353.473,Z 931.342,A -85,B 0,C 180,E1 -13410,E2 -13410} C_VEL
LIN {X 0,Y 353.47,Z 931.276,A -85,B 0,C 180,E1 -13411.139,E2 -13411.139} C_VEL
LIN {X 0,Y 353.369,Z 930.79,A -85,B 0,C 180,E1 -13412.28,E2 -13412.28} C_VEL
LIN {X 0,Y 353.305,Z 929.892,A -85,B 0,C 180,E1 -13413.421,E2 -13413.421} C_VEL
LIN {X 0,Y 353.351,Z 928.536,A -85,B 0,C 180,E1 -13414.563,E2 -13414.563} C_VEL
LIN {X 0,Y 353.392,Z 926.103,A -85,B 0,C 180,E1 -13416.079,E2 -13416.079} C_VEL
LIN {X 0,Y 353.62,Z 921.842,A -85,B 0,C 180,E1 -13417.997,E2 -13417.997} C_VEL
LIN {X 0,Y 354.002,Z 916.85,A -85,B 0,C 180,E1 -13419.715,E2 -13419.715} C_VEL
LIN {X 0,Y 354.781,Z 909.454,A -85,B 0,C 180,E1 -13421.715,E2 -13421.715} C_VEL
LIN {X 0,Y 355.763,Z 901.612,A -85,B 0,C 180,E1 -13423.422,E2 -13423.422} C_VEL
LIN {X 0,Y 356.866,Z 892.548,A -85,B 0,C 180,E1 -13425.028,E2 -13425.028} C_VEL
LIN {X 0,Y 358.187,Z 882.195,A -85,B 0,C 180,E1 -13426.529,E2 -13426.529} C_VEL
LIN {X 0,Y 359.888,Z 870.384,A -85,B 0,C 180,E1 -13427.913,E2 -13427.913} C_VEL
LIN {X 0,Y 360.441,Z 863.481,A -85,B 0,C 180,E1 -13428.62,E2 -13428.62} C_VEL
LIN {X 0,Y 360.134,Z 850.09,A -85,B 0,C 180,E1 -13429.863,E2 -13429.863} C_VEL
LIN {X 0,Y 358.997,Z 839.807,A -85,B 0,C 180,E1 -13430.733,E2 -13430.733} C_VEL
LIN {X 0,Y 356.343,Z 827.174,A -85,B 0,C 180,E1 -13431.748,E2 -13431.748} C_VEL
LIN {X 0,Y 354.486,Z 820.08,A -85,B 0,C 180,E1 -13432.321,E2 -13432.321} C_VEL
LIN {X 0,Y 355.123,Z 813.315,A -85,B 0,C 180,E1 -13435.81,E2 -13435.81} C_VEL
LIN {X 0,Y 355.948,Z 806.388,A -85,B 0,C 180,E1 -13439.684,E2 -13439.684} C_VEL
LIN {X 0,Y 356.843,Z 801.336,A -85,B 0,C 180,E1 -13442.794,E2 -13442.794} C_VEL
LIN {X 0,Y 357.305,Z 798.427,A -85,B 0,C 180,E1 -13444.779,E2 -13444.779} C_VEL
LIN {X 0,Y 357.594,Z 796.371,A -85,B 0,C 180,E1 -13446.311,E2 -13446.311} C_VEL
LIN {X 0,Y 357.534,Z 793.308,A -85,B 0,C 180,E1 -13448.978,E2 -13448.978} C_VEL
LIN {X 0,Y 357.147,Z 790.572,A -85,B 0,C 180,E1 -13451.995,E2 -13451.995} C_VEL
LIN {X 0,Y 356.775,Z 788.433,A -85,B 0,C 180,E1 -13455.166,E2 -13455.166} C_VEL
LIN {X 0,Y 356.475,Z 786.985,A -85,B 0,C 180,E1 -13458.52,E2 -13458.52} C_VEL
LIN {X 0,Y 356.351,Z 786.412,A -85,B 0,C 180,E1 -13460.867,E2 -13460.867} C_VEL
LIN {X 0,Y 356.136,Z 786.2,A -85,B 0,C 180,E1 -13464.008,E2 -13464.008} C_VEL
LIN {X 0,Y 355.931,Z 786.413,A -85,B 0,C 180,E1 -13466.435,E2 -13466.435} C_VEL
LIN {X 0,Y 355.534,Z 787.006,A -85,B 0,C 180,E1 -13469.071,E2 -13469.071} C_VEL
LIN {X 0,Y 355.103,Z 788.341,A -85,B 0,C 180,E1 -13472.951,E2 -13472.951} C_VEL
LIN {X 0,Y 354.744,Z 790.073,A -85,B 0,C 180,E1 -13476.656,E2 -13476.656} C_VEL
LIN {X 0,Y 354.659,Z 790.858,A -85,B 0,C 180,E1 -13477.896,E2 -13477.896} C_VEL
LIN {X 0,Y 355.796,Z 793.747,A -85,B 0,C 180,E1 -13478.185,E2 -13478.185} C_VEL
LIN {X 0,Y 359.998,Z 803.852,A -85,B 0,C 180,E1 -13479.277,E2 -13479.277} C_VEL
LIN {X 0,Y 362.986,Z 814.497,A -85,B 0,C 180,E1 -13480.404,E2 -13480.404} C_VEL
LIN {X 0,Y 363.46,Z 817.504,A -85,B 0,C 180,E1 -13480.714,E2 -13480.714} C_VEL
LIN {X 0,Y 362.122,Z 829.114,A -85,B 0,C 180,E1 -13481.762,E2 -13481.762} C_VEL
LIN {X 0,Y 360.727,Z 840.118,A -85,B 0,C 180,E1 -13483.007,E2 -13483.007} C_VEL
LIN {X 0,Y 359.304,Z 850.043,A -85,B 0,C 180,E1 -13484.397,E2 -13484.397} C_VEL
LIN {X 0,Y 358.06,Z 858.297,A -85,B 0,C 180,E1 -13485.796,E2 -13485.796} C_VEL
LIN {X 0,Y 356.866,Z 866.489,A -85,B 0,C 180,E1 -13487.488,E2 -13487.488} C_VEL
LIN {X 0,Y 355.865,Z 873.061,A -85,B 0,C 180,E1 -13489.185,E2 -13489.185} C_VEL
LIN {X 0,Y 355.116,Z 878.32,A -85,B 0,C 180,E1 -13490.889,E2 -13490.889} C_VEL
LIN {X 0,Y 354.613,Z 881.799,A -85,B 0,C 180,E1 -13492.283,E2 -13492.283} C_VEL
LIN {X 0,Y 353.899,Z 885.564,A -85,B 0,C 180,E1 -13494.3,E2 -13494.3} C_VEL
LIN {X 0,Y 353.934,Z 887.049,A -85,B 0,C 180,E1 -13495.443,E2 -13495.443} C_VEL
LIN {X 0,Y 353.778,Z 888.155,A -85,B 0,C 180,E1 -13496.582,E2 -13496.582} C_VEL
LIN {X 0,Y 353.621,Z 888.821,A -85,B 0,C 180,E1 -13497.721,E2 -13497.721} C_VEL
LIN {X 0,Y 353.521,Z 889.076,A -85,B 0,C 180,E1 -13498.86,E2 -13498.86} C_VEL
LIN {X 0,Y 353.474,Z 888.937,A -85,B 0,C 180,E1 -13499.999,E2 -13499.999} C_VEL
LIN {X 0,Y 353.501,Z 888.395,A -85,B 0,C 180,E1 -13501.138,E2 -13501.138} C_VEL
LIN {X 0,Y 353.546,Z 887.406,A -85,B 0,C 180,E1 -13502.277,E2 -13502.277} C_VEL
LIN {X 0,Y 353.509,Z 886.009,A -85,B 0,C 180,E1 -13503.418,E2 -13503.418} C_VEL
LIN {X 0,Y 353.677,Z 883.095,A -85,B 0,C 180,E1 -13505.129,E2 -13505.129} C_VEL
LIN {X 0,Y 353.978,Z 878.603,A -85,B 0,C 180,E1 -13507.035,E2 -13507.035} C_VEL
LIN {X 0,Y 354.238,Z 874.009,A -85,B 0,C 180,E1 -13508.556,E2 -13508.556} C_VEL
LIN {X 0,Y 354.844,Z 867.592,A -85,B 0,C 180,E1 -13510.267,E2 -13510.267} C_VEL
LIN {X 0,Y 355.55,Z 859.606,A -85,B 0,C 180,E1 -13511.977,E2 -13511.977} C_VEL
LIN {X 0,Y 356.486,Z 849.706,A -85,B 0,C 180,E1 -13513.683,E2 -13513.683} C_VEL
LIN {X 0,Y 357.386,Z 840.119,A -85,B 0,C 180,E1 -13515.025,E2 -13515.025} C_VEL
LIN {X 0,Y 358.314,Z 828.153,A -85,B 0,C 180,E1 -13516.375,E2 -13516.375} C_VEL
LIN {X 0,Y 359.115,Z 817.256,A -85,B 0,C 180,E1 -13517.363,E2 -13517.363} C_VEL
LIN {X 0,Y 359.541,Z 811.751,A -85,B 0,C 180,E1 -13517.782,E2 -13517.782} C_VEL
LIN {X 0,Y 356.706,Z 798.504,A -85,B 0,C 180,E1 -13518.745,E2 -13518.745} C_VEL
LIN {X 0,Y 353.751,Z 785.49,A -85,B 0,C 180,E1 -13519.48,E2 -13519.48} C_VEL
LIN {X 0,Y 353.614,Z 784.583,A -85,B 0,C 180,E1 -13519.545,E2 -13519.545} C_VEL
LIN {X 0,Y 353.733,Z 780.902,A -85,B 0,C 180,E1 -13523.412,E2 -13523.412} C_VEL
LIN {X 0,Y 353.805,Z 777.416,A -85,B 0,C 180,E1 -13527.184,E2 -13527.184} C_VEL
LIN {X 0,Y 354.077,Z 777.379,A -85,B 0,C 180,E1 -13529.749,E2 -13529.749} C_VEL
LIN {X 0,Y 354.442,Z 777.337,A -85,B 0,C 180,E1 -13532.367,E2 -13532.367} C_VEL
LIN {X 0,Y 354.728,Z 777.296,A -85,B 0,C 180,E1 -13535.678,E2 -13535.678} C_VEL
LIN {X 0,Y 354.811,Z 777.286,A -85,B 0,C 180,E1 -13539.333,E2 -13539.333} C_VEL
LIN {X 0,Y 354.783,Z 777.294,A -85,B 0,C 180,E1 -13542.866,E2 -13542.866} C_VEL
LIN {X 0,Y 354.761,Z 777.292,A -85,B 0,C 180,E1 -13546.102,E2 -13546.102} C_VEL
LIN {X 0,Y 354.782,Z 777.292,A -85,B 0,C 180,E1 -13549.178,E2 -13549.178} C_VEL
LIN {X 0,Y 354.8,Z 777.288,A -85,B 0,C 180,E1 -13552.402,E2 -13552.402} C_VEL
LIN {X 0,Y 354.805,Z 777.29,A -85,B 0,C 180,E1 -13554.94,E2 -13554.94} C_VEL
LIN {X 0,Y 354.785,Z 777.289,A -85,B 0,C 180,E1 -13558.404,E2 -13558.404} C_VEL
LIN {X 0,Y 354.794,Z 777.29,A -85,B 0,C 180,E1 -13561.614,E2 -13561.614} C_VEL
LIN {X 0,Y 354.842,Z 777.287,A -85,B 0,C 180,E1 -13565.422,E2 -13565.422} C_VEL
LIN {X 0,Y 354.818,Z 777.287,A -85,B 0,C 180,E1 -13569.113,E2 -13569.113} C_VEL
LIN {X 0,Y 354.871,Z 777.277,A -85,B 0,C 180,E1 -13572.718,E2 -13572.718} C_VEL
LIN {X 0,Y 354.942,Z 777.269,A -85,B 0,C 180,E1 -13576.255,E2 -13576.255} C_VEL
LIN {X 0,Y 354.945,Z 777.274,A -85,B 0,C 180,E1 -13579.735,E2 -13579.735} C_VEL
LIN {X 0,Y 355.075,Z 777.253,A -85,B 0,C 180,E1 -13583.18,E2 -13583.18} C_VEL
LIN {X 0,Y 355.215,Z 777.238,A -85,B 0,C 180,E1 -13587.732,E2 -13587.732} C_VEL
LIN {X 0,Y 355.134,Z 777.244,A -85,B 0,C 180,E1 -13591.134,E2 -13591.134} C_VEL
LIN {X 0,Y 355.208,Z 777.239,A -85,B 0,C 180,E1 -13592.268,E2 -13592.268} C_VEL
LIN {X 0,Y 355.074,Z 777.252,A -85,B 0,C 180,E1 -13596.82,E2 -13596.82} C_VEL
LIN {X 0,Y 354.941,Z 777.275,A -85,B 0,C 180,E1 -13600.265,E2 -13600.265} C_VEL
LIN {X 0,Y 354.934,Z 777.272,A -85,B 0,C 180,E1 -13604.019,E2 -13604.019} C_VEL
LIN {X 0,Y 354.881,Z 777.278,A -85,B 0,C 180,E1 -13608.093,E2 -13608.093} C_VEL
LIN {X 0,Y 354.806,Z 777.287,A -85,B 0,C 180,E1 -13612.108,E2 -13612.108} C_VEL
LIN {X 0,Y 354.84,Z 777.287,A -85,B 0,C 180,E1 -13614.578,E2 -13614.578} C_VEL
LIN {X 0,Y 354.793,Z 777.29,A -85,B 0,C 180,E1 -13618.386,E2 -13618.386} C_VEL
LIN {X 0,Y 354.779,Z 777.29,A -85,B 0,C 180,E1 -13622.334,E2 -13622.334} C_VEL
LIN {X 0,Y 354.815,Z 777.285,A -85,B 0,C 180,E1 -13625.7,E2 -13625.7} C_VEL
LIN {X 0,Y 354.818,Z 777.287,A -85,B 0,C 180,E1 -13629.425,E2 -13629.425} C_VEL
LIN {X 0,Y 354.782,Z 777.292,A -85,B 0,C 180,E1 -13632.868,E2 -13632.868} C_VEL
LIN {X 0,Y 354.762,Z 777.292,A -85,B 0,C 180,E1 -13636.105,E2 -13636.105} C_VEL
LIN {X 0,Y 354.783,Z 777.293,A -85,B 0,C 180,E1 -13639.18,E2 -13639.18} C_VEL
LIN {X 0,Y 354.816,Z 777.285,A -85,B 0,C 180,E1 -13640.538,E2 -13640.538} C_VEL
LIN {X 0,Y 354.206,Z 777.366,A -85,B 0,C 180,E1 -13641.486,E2 -13641.486} C_VEL
LIN {X 0,Y 351.316,Z 777.735,A -85,B 0,C 180,E1 -13643.024,E2 -13643.024} C_VEL
LIN {X 0,Y 348.807,Z 778.047,A -85,B 0,C 180,E1 -13644.269,E2 -13644.269} C_VEL
LIN {X 0,Y 347.703,Z 778.179,A -85,B 0,C 180,E1 -13645.235,E2 -13645.235} C_VEL
LIN {X 0,Y 347.602,Z 778.189,A -85,B 0,C 180,E1 -13645.562,E2 -13645.562} C_VEL
LIN {X 0,Y 347.372,Z 778.213,A -85,B 0,C 180,E1 -13648.264,E2 -13648.264} C_VEL
LIN {X 0,Y 347.04,Z 778.254,A -85,B 0,C 180,E1 -13650.922,E2 -13650.922} C_VEL
LIN {X 0,Y 346.729,Z 778.297,A -85,B 0,C 180,E1 -13653.519,E2 -13653.519} C_VEL
LIN {X 0,Y 346.558,Z 778.722,A -85,B 0,C 180,E1 -13654.796,E2 -13654.796} C_VEL
LIN {X 0,Y 346.547,Z 782.944,A -85,B 0,C 180,E1 -13658.89,E2 -13658.89} C_VEL
LIN {X 0,Y 346.536,Z 784.595,A -85,B 0,C 180,E1 -13660.331,E2 -13660.331} C_VEL
LIN {X 0,Y 349.293,Z 797.168,A -85,B 0,C 180,E1 -13661.028,E2 -13661.028} C_VEL
LIN {X 0,Y 351.862,Z 809.566,A -85,B 0,C 180,E1 -13661.916,E2 -13661.916} C_VEL
LIN {X 0,Y 352.4,Z 813.136,A -85,B 0,C 180,E1 -13662.205,E2 -13662.205} C_VEL
LIN {X 0,Y 351.447,Z 825.797,A -85,B 0,C 180,E1 -13663.295,E2 -13663.295} C_VEL
LIN {X 0,Y 350.619,Z 836.912,A -85,B 0,C 180,E1 -13664.505,E2 -13664.505} C_VEL
LIN {X 0,Y 349.778,Z 846.313,A -85,B 0,C 180,E1 -13665.752,E2 -13665.752} C_VEL
LIN {X 0,Y 348.849,Z 855.312,A -85,B 0,C 180,E1 -13667.198,E2 -13667.198} C_VEL
LIN {X 0,Y 348.055,Z 864.182,A -85,B 0,C 180,E1 -13668.942,E2 -13668.942} C_VEL
LIN {X 0,Y 347.388,Z 871.317,A -85,B 0,C 180,E1 -13670.687,E2 -13670.687} C_VEL
LIN {X 0,Y 346.967,Z 877.023,A -85,B 0,C 180,E1 -13672.436,E2 -13672.436} C_VEL
LIN {X 0,Y 346.685,Z 881.519,A -85,B 0,C 180,E1 -13674.184,E2 -13674.184} C_VEL
LIN {X 0,Y 346.511,Z 883.911,A -85,B 0,C 180,E1 -13675.348,E2 -13675.348} C_VEL
LIN {X 0,Y 346.397,Z 885.848,A -85,B 0,C 180,E1 -13676.512,E2 -13676.512} C_VEL
LIN {X 0,Y 346.439,Z 887.308,A -85,B 0,C 180,E1 -13677.676,E2 -13677.676} C_VEL
LIN {X 0,Y 346.412,Z 888.374,A -85,B 0,C 180,E1 -13678.839,E2 -13678.839} C_VEL
LIN {X 0,Y 346.393,Z 889.037,A -85,B 0,C 180,E1 -13680.001,E2 -13680.001} C_VEL
LIN {X 0,Y 346.449,Z 889.241,A -85,B 0,C 180,E1 -13681.164,E2 -13681.164} C_VEL
LIN {X 0,Y 346.552,Z 889.048,A -85,B 0,C 180,E1 -13682.326,E2 -13682.326} C_VEL
LIN {X 0,Y 346.719,Z 888.46,A -85,B 0,C 180,E1 -13683.487,E2 -13683.487} C_VEL
LIN {X 0,Y 346.808,Z 887.442,A -85,B 0,C 180,E1 -13684.651,E2 -13684.651} C_VEL
LIN {X 0,Y 346.838,Z 886.02,A -85,B 0,C 180,E1 -13685.816,E2 -13685.816} C_VEL
LIN {X 0,Y 347.517,Z 882.736,A -85,B 0,C 180,E1 -13687.713,E2 -13687.713} C_VEL
LIN {X 0,Y 348.095,Z 879.046,A -85,B 0,C 180,E1 -13689.296,E2 -13689.296} C_VEL
LIN {X 0,Y 348.89,Z 873.893,A -85,B 0,C 180,E1 -13691.034,E2 -13691.034} C_VEL
LIN {X 0,Y 349.931,Z 867.464,A -85,B 0,C 180,E1 -13692.764,E2 -13692.764} C_VEL
LIN {X 0,Y 351.214,Z 859.522,A -85,B 0,C 180,E1 -13694.486,E2 -13694.486} C_VEL
LIN {X 0,Y 352.233,Z 853.237,A -85,B 0,C 180,E1 -13695.627,E2 -13695.627} C_VEL
LIN {X 0,Y 353.801,Z 842.728,A -85,B 0,C 180,E1 -13697.201,E2 -13697.201} C_VEL
LIN {X 0,Y 355.221,Z 832.501,A -85,B 0,C 180,E1 -13698.456,E2 -13698.456} C_VEL
LIN {X 0,Y 356.704,Z 821.161,A -85,B 0,C 180,E1 -13699.57,E2 -13699.57} C_VEL
LIN {X 0,Y 357.025,Z 818.295,A -85,B 0,C 180,E1 -13699.822,E2 -13699.822} C_VEL
LIN {X 0,Y 354.856,Z 808.491,A -85,B 0,C 180,E1 -13700.886,E2 -13700.886} C_VEL
LIN {X 0,Y 351.232,Z 798.396,A -85,B 0,C 180,E1 -13702.022,E2 -13702.022} C_VEL
LIN {X 0,Y 348.398,Z 792.175,A -85,B 0,C 180,E1 -13702.734,E2 -13702.734} C_VEL
LIN {X 0,Y 347.58,Z 789.757,A -85,B 0,C 180,E1 -13702.987,E2 -13702.987} C_VEL
LIN {X 0,Y 347.722,Z 786.715,A -85,B 0,C 180,E1 -13706.402,E2 -13706.402} C_VEL
LIN {X 0,Y 347.921,Z 783.331,A -85,B 0,C 180,E1 -13710.332,E2 -13710.332} C_VEL
LIN {X 0,Y 347.967,Z 781.095,A -85,B 0,C 180,E1 -13713.048,E2 -13713.048} C_VEL
LIN {X 0,Y 347.815,Z 778.845,A -85,B 0,C 180,E1 -13716.075,E2 -13716.075} C_VEL
LIN {X 0,Y 347.742,Z 778.17,A -85,B 0,C 180,E1 -13717.324,E2 -13717.324} C_VEL
LIN {X 0,Y 347.736,Z 778.172,A -85,B 0,C 180,E1 -13720.298,E2 -13720.298} C_VEL
LIN {X 0,Y 347.727,Z 778.171,A -85,B 0,C 180,E1 -13723.409,E2 -13723.409} C_VEL
LIN {X 0,Y 347.82,Z 778.388,A -85,B 0,C 180,E1 -13724.601,E2 -13724.601} C_VEL
LIN {X 0,Y 348.883,Z 784.335,A -85,B 0,C 180,E1 -13728.336,E2 -13728.336} C_VEL
LIN {X 0,Y 349.858,Z 789.75,A -85,B 0,C 180,E1 -13731.578,E2 -13731.578} C_VEL
LIN {X 0,Y 350.212,Z 792.91,A -85,B 0,C 180,E1 -13733.391,E2 -13733.391} C_VEL
LIN {X 0,Y 349.883,Z 797.274,A -85,B 0,C 180,E1 -13735.776,E2 -13735.776} C_VEL
LIN {X 0,Y 348.908,Z 804.834,A -85,B 0,C 180,E1 -13739.763,E2 -13739.763} C_VEL
LIN {X 0,Y 348.099,Z 812.342,A -85,B 0,C 180,E1 -13743.629,E2 -13743.629} C_VEL
LIN {X 0,Y 347.471,Z 819.651,A -85,B 0,C 180,E1 -13747.321,E2 -13747.321} C_VEL
LIN {X 0,Y 348.193,Z 823.254,A -85,B 0,C 180,E1 -13747.591,E2 -13747.591} C_VEL
LIN {X 0,Y 350.872,Z 834.598,A -85,B 0,C 180,E1 -13748.547,E2 -13748.547} C_VEL
LIN {X 0,Y 352.57,Z 845.998,A -85,B 0,C 180,E1 -13749.536,E2 -13749.536} C_VEL
LIN {X 0,Y 353.154,Z 861.242,A -85,B 0,C 180,E1 -13750.981,E2 -13750.981} C_VEL
LIN {X 0,Y 353.193,Z 866.796,A -85,B 0,C 180,E1 -13751.585,E2 -13751.585} C_VEL
LIN {X 0,Y 351.682,Z 877.839,A -85,B 0,C 180,E1 -13752.857,E2 -13752.857} C_VEL
LIN {X 0,Y 350.301,Z 887.987,A -85,B 0,C 180,E1 -13754.275,E2 -13754.275} C_VEL
LIN {X 0,Y 348.966,Z 898.051,A -85,B 0,C 180,E1 -13756.015,E2 -13756.015} C_VEL
LIN {X 0,Y 347.912,Z 906.226,A -85,B 0,C 180,E1 -13757.754,E2 -13757.754} C_VEL
LIN {X 0,Y 347.183,Z 912.923,A -85,B 0,C 180,E1 -13759.503,E2 -13759.503} C_VEL
LIN {X 0,Y 346.682,Z 918.297,A -85,B 0,C 180,E1 -13761.255,E2 -13761.255} C_VEL
LIN {X 0,Y 346.419,Z 922.507,A -85,B 0,C 180,E1 -13763.008,E2 -13763.008} C_VEL
LIN {X 0,Y 346.36,Z 926.578,A -85,B 0,C 180,E1 -13765.345,E2 -13765.345} C_VEL
LIN {X 0,Y 346.233,Z 928.294,A -85,B 0,C 180,E1 -13766.509,E2 -13766.509} C_VEL
LIN {X 0,Y 346.35,Z 929.585,A -85,B 0,C 180,E1 -13767.674,E2 -13767.674} C_VEL
LIN {X 0,Y 346.411,Z 930.447,A -85,B 0,C 180,E1 -13768.837,E2 -13768.837} C_VEL
LIN {X 0,Y 346.409,Z 930.869,A -85,B 0,C 180,E1 -13770,E2 -13770} C_VEL
LIN {X 0,Y 346.405,Z 930.832,A -85,B 0,C 180,E1 -13771.163,E2 -13771.163} C_VEL
LIN {X 0,Y 346.273,Z 930.377,A -85,B 0,C 180,E1 -13772.326,E2 -13772.326} C_VEL
LIN {X 0,Y 346.225,Z 929.515,A -85,B 0,C 180,E1 -13773.491,E2 -13773.491} C_VEL
LIN {X 0,Y 346.263,Z 928.219,A -85,B 0,C 180,E1 -13774.657,E2 -13774.657} C_VEL
LIN {X 0,Y 346.287,Z 926.127,A -85,B 0,C 180,E1 -13776.021,E2 -13776.021} C_VEL
LIN {X 0,Y 346.557,Z 921.641,A -85,B 0,C 180,E1 -13778.161,E2 -13778.161} C_VEL
LIN {X 0,Y 346.986,Z 916.754,A -85,B 0,C 180,E1 -13779.914,E2 -13779.914} C_VEL
LIN {X 0,Y 347.809,Z 909.488,A -85,B 0,C 180,E1 -13781.953,E2 -13781.953} C_VEL
LIN {X 0,Y 348.853,Z 901.743,A -85,B 0,C 180,E1 -13783.693,E2 -13783.693} C_VEL
LIN {X 0,Y 349.949,Z 893.39,A -85,B 0,C 180,E1 -13785.246,E2 -13785.246} C_VEL
LIN {X 0,Y 351.42,Z 882.815,A -85,B 0,C 180,E1 -13786.857,E2 -13786.857} C_VEL
LIN {X 0,Y 353.197,Z 871.351,A -85,B 0,C 180,E1 -13788.264,E2 -13788.264} C_VEL
LIN {X 0,Y 353.797,Z 864.61,A -85,B 0,C 180,E1 -13788.983,E2 -13788.983} C_VEL
LIN {X 0,Y 353.66,Z 851.03,A -85,B 0,C 180,E1 -13790.327,E2 -13790.327} C_VEL
LIN {X 0,Y 352.658,Z 841.45,A -85,B 0,C 180,E1 -13791.187,E2 -13791.187} C_VEL
LIN {X 0,Y 350.236,Z 829.44,A -85,B 0,C 180,E1 -13792.244,E2 -13792.244} C_VEL
LIN {X 0,Y 347.576,Z 819.713,A -85,B 0,C 180,E1 -13793.064,E2 -13793.064} C_VEL
LIN {X 0,Y 347.568,Z 819.155,A -85,B 0,C 180,E1 -13793.222,E2 -13793.222} C_VEL
LIN {X 0,Y 348.19,Z 813.314,A -85,B 0,C 180,E1 -13796.363,E2 -13796.363} C_VEL
LIN {X 0,Y 348.994,Z 807.036,A -85,B 0,C 180,E1 -13800.01,E2 -13800.01} C_VEL
LIN {X 0,Y 349.875,Z 802.561,A -85,B 0,C 180,E1 -13802.844,E2 -13802.844} C_VEL
LIN {X 0,Y 350.461,Z 798.771,A -85,B 0,C 180,E1 -13805.56,E2 -13805.56} C_VEL
LIN {X 0,Y 350.647,Z 797.021,A -85,B 0,C 180,E1 -13806.962,E2 -13806.962} C_VEL
LIN {X 0,Y 350.639,Z 795.212,A -85,B 0,C 180,E1 -13808.583,E2 -13808.583} C_VEL
LIN {X 0,Y 350.292,Z 792.538,A -85,B 0,C 180,E1 -13811.46,E2 -13811.46} C_VEL
LIN {X 0,Y 349.927,Z 790.288,A -85,B 0,C 180,E1 -13814.664,E2 -13814.664} C_VEL
LIN {X 0,Y 349.609,Z 788.688,A -85,B 0,C 180,E1 -13818.056,E2 -13818.056} C_VEL
LIN {X 0,Y 349.363,Z 787.864,A -85,B 0,C 180,E1 -13821.418,E2 -13821.418} C_VEL
LIN {X 0,Y 349.174,Z 787.692,A -85,B 0,C 180,E1 -13824.288,E2 -13824.288} C_VEL
LIN {X 0,Y 348.758,Z 788.108,A -85,B 0,C 180,E1 -13827.819,E2 -13827.819} C_VEL
LIN {X 0,Y 348.318,Z 788.971,A -85,B 0,C 180,E1 -13831.036,E2 -13831.036} C_VEL
LIN {X 0,Y 348.047,Z 789.925,A -85,B 0,C 180,E1 -13833.624,E2 -13833.624} C_VEL
LIN {X 0,Y 347.706,Z 791.578,A -85,B 0,C 180,E1 -13837.101,E2 -13837.101} C_VEL
LIN {X 0,Y 348.884,Z 794.615,A -85,B 0,C 180,E1 -13837.432,E2 -13837.432} C_VEL
LIN {X 0,Y 352.878,Z 803.65,A -85,B 0,C 180,E1 -13838.497,E2 -13838.497} C_VEL
LIN {X 0,Y 355.975,Z 813.438,A -85,B 0,C 180,E1 -13839.615,E2 -13839.615} C_VEL
LIN {X 0,Y 357.127,Z 818.639,A -85,B 0,C 180,E1 -13840.203,E2 -13840.203} C_VEL
LIN {X 0,Y 355.615,Z 831.336,A -85,B 0,C 180,E1 -13841.416,E2 -13841.416} C_VEL
LIN {X 0,Y 354.005,Z 842.932,A -85,B 0,C 180,E1 -13842.823,E2 -13842.823} C_VEL
LIN {X 0,Y 352.335,Z 853.36,A -85,B 0,C 180,E1 -13844.377,E2 -13844.377} C_VEL
LIN {X 0,Y 351.071,Z 861.112,A -85,B 0,C 180,E1 -13845.803,E2 -13845.803} C_VEL
LIN {X 0,Y 349.848,Z 868.76,A -85,B 0,C 180,E1 -13847.527,E2 -13847.527} C_VEL
LIN {X 0,Y 348.971,Z 874.053,A -85,B 0,C 180,E1 -13848.969,E2 -13848.969} C_VEL
LIN {X 0,Y 348.174,Z 879.221,A -85,B 0,C 180,E1 -13850.706,E2 -13850.706} C_VEL
LIN {X 0,Y 347.635,Z 882.644,A -85,B 0,C 180,E1 -13852.146,E2 -13852.146} C_VEL
LIN {X 0,Y 346.867,Z 886.255,A -85,B 0,C 180,E1 -13854.184,E2 -13854.184} C_VEL
LIN {X 0,Y 346.895,Z 887.686,A -85,B 0,C 180,E1 -13855.351,E2 -13855.351} C_VEL
LIN {X 0,Y 346.736,Z 888.738,A -85,B 0,C 180,E1 -13856.513,E2 -13856.513} C_VEL
LIN {X 0,Y 346.567,Z 889.347,A -85,B 0,C 180,E1 -13857.674,E2 -13857.674} C_VEL
LIN {X 0,Y 346.459,Z 889.56,A -85,B 0,C 180,E1 -13858.836,E2 -13858.836} C_VEL
LIN {X 0,Y 346.41,Z 889.377,A -85,B 0,C 180,E1 -13859.999,E2 -13859.999} C_VEL
LIN {X 0,Y 346.439,Z 888.765,A -85,B 0,C 180,E1 -13861.161,E2 -13861.161} C_VEL
LIN {X 0,Y 346.452,Z 887.725,A -85,B 0,C 180,E1 -13862.324,E2 -13862.324} C_VEL
LIN {X 0,Y 346.422,Z 886.284,A -85,B 0,C 180,E1 -13863.488,E2 -13863.488} C_VEL
LIN {X 0,Y 346.626,Z 883.287,A -85,B 0,C 180,E1 -13865.234,E2 -13865.234} C_VEL
LIN {X 0,Y 346.91,Z 879.043,A -85,B 0,C 180,E1 -13867.052,E2 -13867.052} C_VEL
LIN {X 0,Y 347.309,Z 873.041,A -85,B 0,C 180,E1 -13869.021,E2 -13869.021} C_VEL
LIN {X 0,Y 347.936,Z 866.256,A -85,B 0,C 180,E1 -13870.767,E2 -13870.767} C_VEL
LIN {X 0,Y 348.7,Z 857.865,A -85,B 0,C 180,E1 -13872.512,E2 -13872.512} C_VEL
LIN {X 0,Y 349.576,Z 849.343,A -85,B 0,C 180,E1 -13873.959,E2 -13873.959} C_VEL
LIN {X 0,Y 350.589,Z 838.361,A -85,B 0,C 180,E1 -13875.474,E2 -13875.474} C_VEL
LIN {X 0,Y 351.441,Z 827.388,A -85,B 0,C 180,E1 -13876.705,E2 -13876.705} C_VEL
LIN {X 0,Y 352.403,Z 814.58,A -85,B 0,C 180,E1 -13877.833,E2 -13877.833} C_VEL
LIN {X 0,Y 352.564,Z 812.823,A -85,B 0,C 180,E1 -13877.968,E2 -13877.968} C_VEL
LIN {X 0,Y 350.043,Z 800.825,A -85,B 0,C 180,E1 -13878.888,E2 -13878.888} C_VEL
LIN {X 0,Y 346.885,Z 786.668,A -85,B 0,C 180,E1 -13879.729,E2 -13879.729} C_VEL
LIN {X 0,Y 346.555,Z 784.97,A -85,B 0,C 180,E1 -13879.817,E2 -13879.817} C_VEL
LIN {X 0,Y 346.674,Z 781.106,A -85,B 0,C 180,E1 -13883.918,E2 -13883.918} C_VEL
LIN {X 0,Y 346.757,Z 778.366,A -85,B 0,C 180,E1 -13886.901,E2 -13886.901} C_VEL
LIN {X 0,Y 347.127,Z 778.248,A -85,B 0,C 180,E1 -13890.406,E2 -13890.406} C_VEL
LIN {X 0,Y 347.559,Z 778.191,A -85,B 0,C 180,E1 -13893.997,E2 -13893.997} C_VEL
LIN {X 0,Y 347.735,Z 778.167,A -85,B 0,C 180,E1 -13897.322,E2 -13897.322} C_VEL
LIN {X 0,Y 347.728,Z 778.171,A -85,B 0,C 180,E1 -13900.296,E2 -13900.296} C_VEL
LIN {X 0,Y 347.718,Z 778.169,A -85,B 0,C 180,E1 -13903.407,E2 -13903.407} C_VEL
LIN {X 0,Y 347.719,Z 778.173,A -85,B 0,C 180,E1 -13906.685,E2 -13906.685} C_VEL
LIN {X 0,Y 347.741,Z 778.166,A -85,B 0,C 180,E1 -13910.172,E2 -13910.172} C_VEL
LIN {X 0,Y 347.755,Z 778.167,A -85,B 0,C 180,E1 -13912.678,E2 -13912.678} C_VEL
LIN {X 0,Y 347.741,Z 778.166,A -85,B 0,C 180,E1 -13915.955,E2 -13915.955} C_VEL
LIN {X 0,Y 347.733,Z 778.168,A -85,B 0,C 180,E1 -13919.65,E2 -13919.65} C_VEL
LIN {X 0,Y 347.747,Z 778.168,A -85,B 0,C 180,E1 -13923.601,E2 -13923.601} C_VEL
LIN {X 0,Y 347.762,Z 778.163,A -85,B 0,C 180,E1 -13926.16,E2 -13926.16} C_VEL
LIN {X 0,Y 347.791,Z 778.161,A -85,B 0,C 180,E1 -13929.908,E2 -13929.908} C_VEL
LIN {X 0,Y 347.823,Z 778.161,A -85,B 0,C 180,E1 -13933.568,E2 -13933.568} C_VEL
LIN {X 0,Y 347.88,Z 778.15,A -85,B 0,C 180,E1 -13937.16,E2 -13937.16} C_VEL
LIN {X 0,Y 347.925,Z 778.142,A -85,B 0,C 180,E1 -13940.7,E2 -13940.7} C_VEL
LIN {X 0,Y 348.026,Z 778.132,A -85,B 0,C 180,E1 -13944.205,E2 -13944.205} C_VEL
LIN {X 0,Y 348.177,Z 778.115,A -85,B 0,C 180,E1 -13947.686,E2 -13947.686} C_VEL
LIN {X 0,Y 348.105,Z 778.12,A -85,B 0,C 180,E1 -13951.157,E2 -13951.157} C_VEL
LIN {X 0,Y 348.169,Z 778.116,A -85,B 0,C 180,E1 -13952.314,E2 -13952.314} C_VEL
LIN {X 0,Y 348.042,Z 778.128,A -85,B 0,C 180,E1 -13956.959,E2 -13956.959} C_VEL
LIN {X 0,Y 347.881,Z 778.152,A -85,B 0,C 180,E1 -13960.476,E2 -13960.476} C_VEL
LIN {X 0,Y 347.89,Z 778.151,A -85,B 0,C 180,E1 -13964.15,E2 -13964.15} C_VEL
LIN {X 0,Y 347.82,Z 778.159,A -85,B 0,C 180,E1 -13968.26,E2 -13968.26} C_VEL
LIN {X 0,Y 347.759,Z 778.163,A -85,B 0,C 180,E1 -13971.627,E2 -13971.627} C_VEL
LIN {X 0,Y 347.761,Z 778.165,A -85,B 0,C 180,E1 -13975.113,E2 -13975.113} C_VEL
LIN {X 0,Y 347.729,Z 778.167,A -85,B 0,C 180,E1 -13977.701,E2 -13977.701} C_VEL
LIN {X 0,Y 347.733,Z 778.168,A -85,B 0,C 180,E1 -13980.35,E2 -13980.35} C_VEL
LIN {X 0,Y 347.741,Z 778.166,A -85,B 0,C 180,E1 -13984.045,E2 -13984.045} C_VEL
LIN {X 0,Y 347.755,Z 778.167,A -85,B 0,C 180,E1 -13987.322,E2 -13987.322} C_VEL
LIN {X 0,Y 347.726,Z 778.168,A -85,B 0,C 180,E1 -13990.298,E2 -13990.298} C_VEL
LIN {X 0,Y 347.717,Z 778.173,A -85,B 0,C 180,E1 -13993.409,E2 -13993.409} C_VEL
LIN {X 0,Y 347.72,Z 778.169,A -85,B 0,C 180,E1 -13996.688,E2 -13996.688} C_VEL
LIN {X 0,Y 347.743,Z 778.166,A -85,B 0,C 180,E1 -14000.174,E2 -14000.174} C_VEL
LIN {X 0,Y 347.736,Z 778.167,A -85,B 0,C 180,E1 -14002.678,E2 -14002.678} C_VEL
LIN {X 0,Y 347.602,Z 778.189,A -85,B 0,C 180,E1 -14005.562,E2 -14005.562} C_VEL
LIN {X 0,Y 346.875,Z 778.274,A -85,B 0,C 180,E1 -14006.528,E2 -14006.528} C_VEL
LIN {X 0,Y 343.869,Z 778.65,A -85,B 0,C 180,E1 -14008.094,E2 -14008.094} C_VEL
LIN {X 0,Y 341.291,Z 778.973,A -85,B 0,C 180,E1 -14009.362,E2 -14009.362} C_VEL
LIN {X 0,Y 340.121,Z 779.116,A -85,B 0,C 180,E1 -14010.346,E2 -14010.346} C_VEL
LIN {X 0,Y 339.991,Z 779.131,A -85,B 0,C 180,E1 -14010.681,E2 -14010.681} C_VEL
LIN {X 0,Y 339.559,Z 779.19,A -85,B 0,C 180,E1 -14014.239,E2 -14014.239} C_VEL
LIN {X 0,Y 339.435,Z 781.486,A -85,B 0,C 180,E1 -14016.836,E2 -14016.836} C_VEL
LIN {X 0,Y 339.448,Z 784.799,A -85,B 0,C 180,E1 -14020.027,E2 -14020.027} C_VEL
LIN {X 0,Y 342.822,Z 800.563,A -85,B 0,C 180,E1 -14020.966,E2 -14020.966} C_VEL
LIN {X 0,Y 345.268,Z 812.445,A -85,B 0,C 180,E1 -14021.879,E2 -14021.879} C_VEL
LIN {X 0,Y 345.235,Z 816.657,A -85,B 0,C 180,E1 -14022.222,E2 -14022.222} C_VEL
LIN {X 0,Y 344.361,Z 827.782,A -85,B 0,C 180,E1 -14023.247,E2 -14023.247} C_VEL
LIN {X 0,Y 343.436,Z 839.267,A -85,B 0,C 180,E1 -14024.573,E2 -14024.573} C_VEL
LIN {X 0,Y 342.438,Z 849.604,A -85,B 0,C 180,E1 -14026.047,E2 -14026.047} C_VEL
LIN {X 0,Y 341.606,Z 858.146,A -85,B 0,C 180,E1 -14027.526,E2 -14027.526} C_VEL
LIN {X 0,Y 340.827,Z 866.501,A -85,B 0,C 180,E1 -14029.306,E2 -14029.306} C_VEL
LIN {X 0,Y 340.154,Z 873.272,A -85,B 0,C 180,E1 -14031.087,E2 -14031.087} C_VEL
LIN {X 0,Y 339.751,Z 879.498,A -85,B 0,C 180,E1 -14033.178,E2 -14033.178} C_VEL
LIN {X 0,Y 339.453,Z 884.078,A -85,B 0,C 180,E1 -14035.251,E2 -14035.251} C_VEL
LIN {X 0,Y 339.317,Z 886.089,A -85,B 0,C 180,E1 -14036.439,E2 -14036.439} C_VEL
LIN {X 0,Y 339.344,Z 887.61,A -85,B 0,C 180,E1 -14037.627,E2 -14037.627} C_VEL
LIN {X 0,Y 339.334,Z 888.721,A -85,B 0,C 180,E1 -14038.814,E2 -14038.814} C_VEL
LIN {X 0,Y 339.332,Z 889.435,A -85,B 0,C 180,E1 -14040.001,E2 -14040.001} C_VEL
LIN {X 0,Y 339.389,Z 889.711,A -85,B 0,C 180,E1 -14041.188,E2 -14041.188} C_VEL
LIN {X 0,Y 339.675,Z 889.023,A -85,B 0,C 180,E1 -14043.56,E2 -14043.56} C_VEL
LIN {X 0,Y 339.759,Z 888.096,A -85,B 0,C 180,E1 -14044.747,E2 -14044.747} C_VEL
LIN {X 0,Y 339.811,Z 886.723,A -85,B 0,C 180,E1 -14045.937,E2 -14045.937} C_VEL
LIN {X 0,Y 340.521,Z 883.603,A -85,B 0,C 180,E1 -14047.831,E2 -14047.831} C_VEL
LIN {X 0,Y 341.419,Z 878.404,A -85,B 0,C 180,E1 -14050.078,E2 -14050.078} C_VEL
LIN {X 0,Y 342.491,Z 871.954,A -85,B 0,C 180,E1 -14052.143,E2 -14052.143} C_VEL
LIN {X 0,Y 343.768,Z 864.976,A -85,B 0,C 180,E1 -14053.9,E2 -14053.9} C_VEL
LIN {X 0,Y 345.224,Z 856.321,A -85,B 0,C 180,E1 -14055.65,E2 -14055.65} C_VEL
LIN {X 0,Y 347.063,Z 845.713,A -85,B 0,C 180,E1 -14057.378,E2 -14057.378} C_VEL
LIN {X 0,Y 348.517,Z 835.981,A -85,B 0,C 180,E1 -14058.659,E2 -14058.659} C_VEL
LIN {X 0,Y 350.286,Z 823.81,A -85,B 0,C 180,E1 -14059.944,E2 -14059.944} C_VEL
LIN {X 0,Y 350.71,Z 820.323,A -85,B 0,C 180,E1 -14060.258,E2 -14060.258} C_VEL
LIN {X 0,Y 348.996,Z 811.809,A -85,B 0,C 180,E1 -14061.254,E2 -14061.254} C_VEL
LIN {X 0,Y 345.561,Z 801.755,A -85,B 0,C 180,E1 -14062.461,E2 -14062.461} C_VEL
LIN {X 0,Y 341.857,Z 793.546,A -85,B 0,C 180,E1 -14063.493,E2 -14063.493} C_VEL
LIN {X 0,Y 340.686,Z 790.451,A -85,B 0,C 180,E1 -14063.882,E2 -14063.882} C_VEL
LIN {X 0,Y 340.877,Z 787.314,A -85,B 0,C 180,E1 -14067.557,E2 -14067.557} C_VEL
LIN {X 0,Y 341.057,Z 784.475,A -85,B 0,C 180,E1 -14071.009,E2 -14071.009} C_VEL
LIN {X 0,Y 341.115,Z 781.866,A -85,B 0,C 180,E1 -14074.5,E2 -14074.5} C_VEL
LIN {X 0,Y 340.959,Z 780.392,A -85,B 0,C 180,E1 -14076.711,E2 -14076.711} C_VEL
LIN {X 0,Y 340.7,Z 779.046,A -85,B 0,C 180,E1 -14079.384,E2 -14079.384} C_VEL
LIN {X 0,Y 340.68,Z 779.051,A -85,B 0,C 180,E1 -14082.905,E2 -14082.905} C_VEL
LIN {X 0,Y 340.738,Z 779.225,A -85,B 0,C 180,E1 -14084.315,E2 -14084.315} C_VEL
LIN {X 0,Y 341.737,Z 784.56,A -85,B 0,C 180,E1 -14087.763,E2 -14087.763} C_VEL
LIN {X 0,Y 342.713,Z 790.155,A -85,B 0,C 180,E1 -14091.195,E2 -14091.195} C_VEL
LIN {X 0,Y 343.195,Z 793.21,A -85,B 0,C 180,E1 -14093.003,E2 -14093.003} C_VEL
LIN {X 0,Y 342.839,Z 798.06,A -85,B 0,C 180,E1 -14095.718,E2 -14095.718} C_VEL
LIN {X 0,Y 341.859,Z 805.449,A -85,B 0,C 180,E1 -14099.707,E2 -14099.707} C_VEL
LIN {X 0,Y 341.019,Z 813.016,A -85,B 0,C 180,E1 -14103.699,E2 -14103.699} C_VEL
LIN {X 0,Y 340.539,Z 818.289,A -85,B 0,C 180,E1 -14106.431,E2 -14106.431} C_VEL
LIN {X 0,Y 341.328,Z 822.131,A -85,B 0,C 180,E1 -14106.74,E2 -14106.74} C_VEL
LIN {X 0,Y 344.228,Z 833.962,A -85,B 0,C 180,E1 -14107.815,E2 -14107.815} C_VEL
LIN {X 0,Y 346.068,Z 846.304,A -85,B 0,C 180,E1 -14108.967,E2 -14108.967} C_VEL
LIN {X 0,Y 346.574,Z 859.81,A -85,B 0,C 180,E1 -14110.298,E2 -14110.298} C_VEL
LIN {X 0,Y 346.543,Z 867.918,A -85,B 0,C 180,E1 -14111.219,E2 -14111.219} C_VEL
LIN {X 0,Y 344.96,Z 878.69,A -85,B 0,C 180,E1 -14112.512,E2 -14112.512} C_VEL
LIN {X 0,Y 343.484,Z 888.585,A -85,B 0,C 180,E1 -14113.966,E2 -14113.966} C_VEL
LIN {X 0,Y 342.093,Z 898.327,A -85,B 0,C 180,E1 -14115.728,E2 -14115.728} C_VEL
LIN {X 0,Y 340.955,Z 906.377,A -85,B 0,C 180,E1 -14117.5,E2 -14117.5} C_VEL
LIN {X 0,Y 340.166,Z 912.898,A -85,B 0,C 180,E1 -14119.284,E2 -14119.284} C_VEL
LIN {X 0,Y 339.65,Z 918.154,A -85,B 0,C 180,E1 -14121.072,E2 -14121.072} C_VEL
LIN {X 0,Y 339.346,Z 922.289,A -85,B 0,C 180,E1 -14122.862,E2 -14122.862} C_VEL
LIN {X 0,Y 339.262,Z 924.454,A -85,B 0,C 180,E1 -14124.055,E2 -14124.055} C_VEL
LIN {X 0,Y 339.16,Z 927.676,A -85,B 0,C 180,E1 -14126.436,E2 -14126.436} C_VEL
LIN {X 0,Y 339.258,Z 928.994,A -85,B 0,C 180,E1 -14127.625,E2 -14127.625} C_VEL
